LIN {X 0,Y 143.393,Z 441.137,A -85,B 0,C 180,E1 -24501.373,E2 -24501.373} C_VEL
LIN {X 0,Y 143.569,Z 442.834,A -85,B 0,C 180,E1 -24508.221,E2 -24508.221} C_VEL
LIN {X 0,Y 143.67,Z 443.783,A -85,B 0,C 180,E1 -24510.704,E2 -24510.704} C_VEL
LIN {X 0,Y 144.829,Z 446.872,A -85,B 0,C 180,E1 -24511.853,E2 -24511.853} C_VEL
LIN {X 0,Y 147.407,Z 450.098,A -85,B 0,C 180,E1 -24513.922,E2 -24513.922} C_VEL
LIN {X 0,Y 149.008,Z 453.626,A -85,B 0,C 180,E1 -24515.399,E2 -24515.399} C_VEL
LIN {X 0,Y 150.515,Z 455.827,A -85,B 0,C 180,E1 -24516.538,E2 -24516.538} C_VEL
LIN {X 0,Y 154.839,Z 465.074,A -85,B 0,C 180,E1 -24520.302,E2 -24520.302} C_VEL
LIN {X 0,Y 156.776,Z 470.615,A -85,B 0,C 180,E1 -24522.256,E2 -24522.256} C_VEL
LIN {X 0,Y 158.409,Z 477.402,A -85,B 0,C 180,E1 -24524.42,E2 -24524.42} C_VEL
LIN {X 0,Y 159.626,Z 487.108,A -85,B 0,C 180,E1 -24527.387,E2 -24527.387} C_VEL
LIN {X 0,Y 159.828,Z 498.246,A -85,B 0,C 180,E1 -24530.923,E2 -24530.923} C_VEL
LIN {X 0,Y 159.156,Z 506.693,A -85,B 0,C 180,E1 -24533.798,E2 -24533.798} C_VEL
LIN {X 0,Y 158.051,Z 513.314,A -85,B 0,C 180,E1 -24536.232,E2 -24536.232} C_VEL
LIN {X 0,Y 154.438,Z 521.15,A -85,B 0,C 180,E1 -24539.206,E2 -24539.206} C_VEL
LIN {X 0,Y 151.218,Z 527.693,A -85,B 0,C 180,E1 -24542.305,E2 -24542.305} C_VEL
LIN {X 0,Y 148.827,Z 532.196,A -85,B 0,C 180,E1 -24544.849,E2 -24544.849} C_VEL
LIN {X 0,Y 145.787,Z 537.691,A -85,B 0,C 180,E1 -24548.804,E2 -24548.804} C_VEL
LIN {X 0,Y 143.393,Z 542.02,A -85,B 0,C 180,E1 -24552.898,E2 -24552.898} C_VEL
LIN {X 0,Y 142.296,Z 544.395,A -85,B 0,C 180,E1 -24555.703,E2 -24555.703} C_VEL
LIN {X 0,Y 141.449,Z 546.201,A -85,B 0,C 180,E1 -24558.536,E2 -24558.536} C_VEL
LIN {X 0,Y 140.624,Z 548.663,A -85,B 0,C 180,E1 -24564.263,E2 -24564.263} C_VEL
LIN {X 0,Y 140.572,Z 549.418,A -85,B 0,C 180,E1 -24569.355,E2 -24569.355} C_VEL
LIN {X 0,Y 140.512,Z 549.259,A -85,B 0,C 180,E1 -24572.866,E2 -24572.866} C_VEL
LIN {X 0,Y 140.623,Z 548.664,A -85,B 0,C 180,E1 -24575.736,E2 -24575.736} C_VEL
LIN {X 0,Y 141.449,Z 546.201,A -85,B 0,C 180,E1 -24581.463,E2 -24581.463} C_VEL
LIN {X 0,Y 142.829,Z 543.242,A -85,B 0,C 180,E1 -24585.701,E2 -24585.701} C_VEL
LIN {X 0,Y 144.915,Z 539.247,A -85,B 0,C 180,E1 -24589.844,E2 -24589.844} C_VEL
LIN {X 0,Y 147.71,Z 534.114,A -85,B 0,C 180,E1 -24593.854,E2 -24593.854} C_VEL
LIN {X 0,Y 150.632,Z 528.852,A -85,B 0,C 180,E1 -24597.058,E2 -24597.058} C_VEL
LIN {X 0,Y 153.161,Z 523.745,A -85,B 0,C 180,E1 -24599.644,E2 -24599.644} C_VEL
LIN {X 0,Y 156.671,Z 516.577,A -85,B 0,C 180,E1 -24602.567,E2 -24602.567} C_VEL
LIN {X 0,Y 158.059,Z 513.317,A -85,B 0,C 180,E1 -24603.765,E2 -24603.765} C_VEL
LIN {X 0,Y 159.429,Z 504.825,A -85,B 0,C 180,E1 -24606.879,E2 -24606.879} C_VEL
LIN {X 0,Y 159.896,Z 494.943,A -85,B 0,C 180,E1 -24610.153,E2 -24610.153} C_VEL
LIN {X 0,Y 159.424,Z 485.143,A -85,B 0,C 180,E1 -24613.195,E2 -24613.195} C_VEL
LIN {X 0,Y 158.141,Z 476.083,A -85,B 0,C 180,E1 -24615.973,E2 -24615.973} C_VEL
LIN {X 0,Y 156.287,Z 468.906,A -85,B 0,C 180,E1 -24618.338,E2 -24618.338} C_VEL
LIN {X 0,Y 154.102,Z 463.522,A -85,B 0,C 180,E1 -24620.319,E2 -24620.319} C_VEL
LIN {X 0,Y 149.931,Z 454.821,A -85,B 0,C 180,E1 -24623.922,E2 -24623.922} C_VEL
LIN {X 0,Y 147.879,Z 451.476,A -85,B 0,C 180,E1 -24625.576,E2 -24625.576} C_VEL
LIN {X 0,Y 147.011,Z 449.414,A -85,B 0,C 180,E1 -24626.424,E2 -24626.424} C_VEL
LIN {X 0,Y 144.642,Z 446.551,A -85,B 0,C 180,E1 -24628.305,E2 -24628.305} C_VEL
LIN {X 0,Y 143.604,Z 443.405,A -85,B 0,C 180,E1 -24629.484,E2 -24629.484} C_VEL
LIN {X 0,Y 143.603,Z 443.398,A -85,B 0,C 180,E1 -24629.509,E2 -24629.509} C_VEL
LIN {X 0,Y 143.264,Z 443.023,A -85,B 0,C 180,E1 -24631.065,E2 -24631.065} C_VEL
LIN {X 0,Y 141.909,Z 442.618,A -85,B 0,C 180,E1 -24633.375,E2 -24633.375} C_VEL
LIN {X 0,Y 136.677,Z 441.804,A -85,B 0,C 180,E1 -24640.485,E2 -24640.485} C_VEL
LIN {X 0,Y 136.28,Z 441.543,A -85,B 0,C 180,E1 -24642.161,E2 -24642.161} C_VEL
LIN {X 0,Y 136.272,Z 441.029,A -85,B 0,C 180,E1 -24645.055,E2 -24645.055} C_VEL
LIN {X 0,Y 136.495,Z 440.983,A -85,B 0,C 180,E1 -24648.113,E2 -24648.113} C_VEL
LIN {X 0,Y 136.597,Z 440.97,A -85,B 0,C 180,E1 -24651.119,E2 -24651.119} C_VEL
LIN {X 0,Y 137.131,Z 440.87,A -85,B 0,C 180,E1 -24659.998,E2 -24659.998} C_VEL
LIN {X 0,Y 136.588,Z 440.963,A -85,B 0,C 180,E1 -24668.878,E2 -24668.878} C_VEL
LIN {X 0,Y 136.488,Z 440.983,A -85,B 0,C 180,E1 -24671.953,E2 -24671.953} C_VEL
LIN {X 0,Y 136.24,Z 441.013,A -85,B 0,C 180,E1 -24678.028,E2 -24678.028} C_VEL
LIN {X 0,Y 136.193,Z 441.017,A -85,B 0,C 180,E1 -24681.747,E2 -24681.747} C_VEL
LIN {X 0,Y 136.082,Z 441.071,A -85,B 0,C 180,E1 -24685.013,E2 -24685.013} C_VEL
LIN {X 0,Y 136.847,Z 443.396,A -85,B 0,C 180,E1 -24686.085,E2 -24686.085} C_VEL
LIN {X 0,Y 138.886,Z 445.821,A -85,B 0,C 180,E1 -24688.301,E2 -24688.301} C_VEL
LIN {X 0,Y 140.192,Z 446.89,A -85,B 0,C 180,E1 -24689.52,E2 -24689.52} C_VEL
LIN {X 0,Y 141.597,Z 449.723,A -85,B 0,C 180,E1 -24691.096,E2 -24691.096} C_VEL
LIN {X 0,Y 143.682,Z 451.967,A -85,B 0,C 180,E1 -24692.892,E2 -24692.892} C_VEL
LIN {X 0,Y 145.815,Z 455.547,A -85,B 0,C 180,E1 -24694.981,E2 -24694.981} C_VEL
LIN {X 0,Y 149.78,Z 462.277,A -85,B 0,C 180,E1 -24698.598,E2 -24698.598} C_VEL
LIN {X 0,Y 153.726,Z 470.155,A -85,B 0,C 180,E1 -24702.4,E2 -24702.4} C_VEL
LIN {X 0,Y 156.806,Z 478.027,A -85,B 0,C 180,E1 -24705.815,E2 -24705.815} C_VEL
LIN {X 0,Y 158.958,Z 485.07,A -85,B 0,C 180,E1 -24708.729,E2 -24708.729} C_VEL
LIN {X 0,Y 160.498,Z 491.796,A -85,B 0,C 180,E1 -24711.465,E2 -24711.465} C_VEL
LIN {X 0,Y 161.573,Z 498.214,A -85,B 0,C 180,E1 -24714.117,E2 -24714.117} C_VEL
LIN {X 0,Y 162.598,Z 505.476,A -85,B 0,C 180,E1 -24717.364,E2 -24717.364} C_VEL
LIN {X 0,Y 164.659,Z 513.088,A -85,B 0,C 180,E1 -24721.399,E2 -24721.399} C_VEL
LIN {X 0,Y 167.754,Z 519.177,A -85,B 0,C 180,E1 -24725.233,E2 -24725.233} C_VEL
LIN {X 0,Y 172.51,Z 524.998,A -85,B 0,C 180,E1 -24729.552,E2 -24729.552} C_VEL
LIN {X 0,Y 176.829,Z 528.462,A -85,B 0,C 180,E1 -24732.525,E2 -24732.525} C_VEL
LIN {X 0,Y 184.325,Z 532.617,A -85,B 0,C 180,E1 -24736.776,E2 -24736.776} C_VEL
LIN {X 0,Y 192.376,Z 535.547,A -85,B 0,C 180,E1 -24740.526,E2 -24740.526} C_VEL
LIN {X 0,Y 201.039,Z 537.521,A -85,B 0,C 180,E1 -24743.981,E2 -24743.981} C_VEL
LIN {X 0,Y 206.856,Z 538.379,A -85,B 0,C 180,E1 -24746.104,E2 -24746.104} C_VEL
LIN {X 0,Y 212.283,Z 538.785,A -85,B 0,C 180,E1 -24748.103,E2 -24748.103} C_VEL
LIN {X 0,Y 216.488,Z 538.826,A -85,B 0,C 180,E1 -24750,E2 -24750} C_VEL
LIN {X 0,Y 212.31,Z 538.784,A -85,B 0,C 180,E1 -24751.897,E2 -24751.897} C_VEL
LIN {X 0,Y 204.513,Z 538.092,A -85,B 0,C 180,E1 -24754.759,E2 -24754.759} C_VEL
LIN {X 0,Y 195.316,Z 536.345,A -85,B 0,C 180,E1 -24758.276,E2 -24758.276} C_VEL
LIN {X 0,Y 186.807,Z 533.661,A -85,B 0,C 180,E1 -24762.003,E2 -24762.003} C_VEL
LIN {X 0,Y 179.372,Z 530.065,A -85,B 0,C 180,E1 -24765.919,E2 -24765.919} C_VEL
LIN {X 0,Y 173.655,Z 526.039,A -85,B 0,C 180,E1 -24769.596,E2 -24769.596} C_VEL
LIN {X 0,Y 168.811,Z 520.752,A -85,B 0,C 180,E1 -24773.668,E2 -24773.668} C_VEL
LIN {X 0,Y 165.747,Z 515.636,A -85,B 0,C 180,E1 -24777.075,E2 -24777.075} C_VEL
LIN {X 0,Y 163.456,Z 509.289,A -85,B 0,C 180,E1 -24780.695,E2 -24780.695} C_VEL
LIN {X 0,Y 162.22,Z 503.336,A -85,B 0,C 180,E1 -24783.649,E2 -24783.649} C_VEL
LIN {X 0,Y 161.234,Z 495.681,A -85,B 0,C 180,E1 -24786.939,E2 -24786.939} C_VEL
LIN {X 0,Y 159.656,Z 487.905,A -85,B 0,C 180,E1 -24790.155,E2 -24790.155} C_VEL
LIN {X 0,Y 157.146,Z 479.075,A -85,B 0,C 180,E1 -24793.77,E2 -24793.77} C_VEL
LIN {X 0,Y 153.7,Z 470.237,A -85,B 0,C 180,E1 -24797.591,E2 -24797.591} C_VEL
LIN {X 0,Y 148.933,Z 460.739,A -85,B 0,C 180,E1 -24802.162,E2 -24802.162} C_VEL
LIN {X 0,Y 145.766,Z 455.541,A -85,B 0,C 180,E1 -24805.049,E2 -24805.049} C_VEL
LIN {X 0,Y 143.589,Z 451.797,A -85,B 0,C 180,E1 -24807.198,E2 -24807.198} C_VEL
LIN {X 0,Y 140.934,Z 448.683,A -85,B 0,C 180,E1 -24809.573,E2 -24809.573} C_VEL
LIN {X 0,Y 140.071,Z 446.555,A -85,B 0,C 180,E1 -24810.64,E2 -24810.64} C_VEL
LIN {X 0,Y 137.435,Z 444.32,A -85,B 0,C 180,E1 -24813.217,E2 -24813.217} C_VEL
LIN {X 0,Y 136.247,Z 441.933,A -85,B 0,C 180,E1 -24814.714,E2 -24814.714} C_VEL
LIN {X 0,Y 136.085,Z 441.023,A -85,B 0,C 180,E1 -24815.09,E2 -24815.09} C_VEL
LIN {X 0,Y 136.242,Z 441.007,A -85,B 0,C 180,E1 -24818.835,E2 -24818.835} C_VEL
LIN {X 0,Y 136.275,Z 440.999,A -85,B 0,C 180,E1 -24825.059,E2 -24825.059} C_VEL
LIN {X 0,Y 136.497,Z 440.982,A -85,B 0,C 180,E1 -24828.116,E2 -24828.116} C_VEL
LIN {X 0,Y 136.591,Z 440.963,A -85,B 0,C 180,E1 -24831.122,E2 -24831.122} C_VEL
LIN {X 0,Y 137.134,Z 440.87,A -85,B 0,C 180,E1 -24840.002,E2 -24840.002} C_VEL
LIN {X 0,Y 136.6,Z 440.97,A -85,B 0,C 180,E1 -24848.881,E2 -24848.881} C_VEL
LIN {X 0,Y 136.492,Z 440.986,A -85,B 0,C 180,E1 -24851.956,E2 -24851.956} C_VEL
LIN {X 0,Y 136.275,Z 441.029,A -85,B 0,C 180,E1 -24854.945,E2 -24854.945} C_VEL
LIN {X 0,Y 136.389,Z 442.204,A -85,B 0,C 180,E1 -24861.145,E2 -24861.145} C_VEL
LIN {X 0,Y 136.395,Z 443.172,A -85,B 0,C 180,E1 -24865.057,E2 -24865.057} C_VEL
LIN {X 0,Y 137.556,Z 446.287,A -85,B 0,C 180,E1 -24866.557,E2 -24866.557} C_VEL
LIN {X 0,Y 140.112,Z 449.358,A -85,B 0,C 180,E1 -24869.122,E2 -24869.122} C_VEL
LIN {X 0,Y 140.609,Z 450.141,A -85,B 0,C 180,E1 -24869.639,E2 -24869.639} C_VEL
LIN {X 0,Y 142.08,Z 453.455,A -85,B 0,C 180,E1 -24871.293,E2 -24871.293} C_VEL
LIN {X 0,Y 143.832,Z 455.753,A -85,B 0,C 180,E1 -24872.826,E2 -24872.826} C_VEL
LIN {X 0,Y 145.538,Z 459.421,A -85,B 0,C 180,E1 -24874.571,E2 -24874.571} C_VEL
LIN {X 0,Y 146.291,Z 460.539,A -85,B 0,C 180,E1 -24875.244,E2 -24875.244} C_VEL
LIN {X 0,Y 150.353,Z 470.127,A -85,B 0,C 180,E1 -24879.437,E2 -24879.437} C_VEL
LIN {X 0,Y 152.33,Z 476.964,A -85,B 0,C 180,E1 -24881.992,E2 -24881.992} C_VEL
LIN {X 0,Y 153.471,Z 485.376,A -85,B 0,C 180,E1 -24884.816,E2 -24884.816} C_VEL
LIN {X 0,Y 153.84,Z 493.755,A -85,B 0,C 180,E1 -24887.61,E2 -24887.61} C_VEL
LIN {X 0,Y 153.408,Z 503.934,A -85,B 0,C 180,E1 -24891.154,E2 -24891.154} C_VEL
LIN {X 0,Y 151.957,Z 513.094,A -85,B 0,C 180,E1 -24894.681,E2 -24894.681} C_VEL
LIN {X 0,Y 150.705,Z 516.362,A -85,B 0,C 180,E1 -24895.971,E2 -24895.971} C_VEL
LIN {X 0,Y 147.619,Z 522.314,A -85,B 0,C 180,E1 -24898.419,E2 -24898.419} C_VEL
LIN {X 0,Y 144.306,Z 528.638,A -85,B 0,C 180,E1 -24901.651,E2 -24901.651} C_VEL
LIN {X 0,Y 141.222,Z 533.9,A -85,B 0,C 180,E1 -24904.975,E2 -24904.975} C_VEL
LIN {X 0,Y 138.221,Z 539.034,A -85,B 0,C 180,E1 -24909.15,E2 -24909.15} C_VEL
LIN {X 0,Y 135.961,Z 543.029,A -85,B 0,C 180,E1 -24913.482,E2 -24913.482} C_VEL
LIN {X 0,Y 134.481,Z 545.989,A -85,B 0,C 180,E1 -24917.933,E2 -24917.933} C_VEL
LIN {X 0,Y 133.55,Z 548.452,A -85,B 0,C 180,E1 -24923.958,E2 -24923.958} C_VEL
LIN {X 0,Y 133.414,Z 549.047,A -85,B 0,C 180,E1 -24926.98,E2 -24926.98} C_VEL
LIN {X 0,Y 133.505,Z 549.208,A -85,B 0,C 180,E1 -24929.999,E2 -24929.999} C_VEL
LIN {X 0,Y 133.415,Z 549.048,A -85,B 0,C 180,E1 -24933.019,E2 -24933.019} C_VEL
LIN {X 0,Y 133.55,Z 548.452,A -85,B 0,C 180,E1 -24936.041,E2 -24936.041} C_VEL
LIN {X 0,Y 134.481,Z 545.989,A -85,B 0,C 180,E1 -24942.065,E2 -24942.065} C_VEL
LIN {X 0,Y 135.96,Z 543.03,A -85,B 0,C 180,E1 -24946.516,E2 -24946.516} C_VEL
LIN {X 0,Y 138.219,Z 539.035,A -85,B 0,C 180,E1 -24950.849,E2 -24950.849} C_VEL
LIN {X 0,Y 141.216,Z 533.901,A -85,B 0,C 180,E1 -24955.025,E2 -24955.025} C_VEL
LIN {X 0,Y 144.308,Z 528.64,A -85,B 0,C 180,E1 -24958.348,E2 -24958.348} C_VEL
LIN {X 0,Y 147.617,Z 522.316,A -85,B 0,C 180,E1 -24961.58,E2 -24961.58} C_VEL
LIN {X 0,Y 150.703,Z 516.365,A -85,B 0,C 180,E1 -24964.028,E2 -24964.028} C_VEL
LIN {X 0,Y 151.961,Z 513.096,A -85,B 0,C 180,E1 -24965.316,E2 -24965.316} C_VEL
LIN {X 0,Y 153.432,Z 503.887,A -85,B 0,C 180,E1 -24968.857,E2 -24968.857} C_VEL
LIN {X 0,Y 153.833,Z 493.811,A -85,B 0,C 180,E1 -24972.374,E2 -24972.374} C_VEL
LIN {X 0,Y 153.466,Z 485.366,A -85,B 0,C 180,E1 -24975.188,E2 -24975.188} C_VEL
LIN {X 0,Y 152.317,Z 477.003,A -85,B 0,C 180,E1 -24978.004,E2 -24978.004} C_VEL
LIN {X 0,Y 150.358,Z 470.111,A -85,B 0,C 180,E1 -24980.565,E2 -24980.565} C_VEL
LIN {X 0,Y 146.266,Z 460.462,A -85,B 0,C 180,E1 -24984.787,E2 -24984.787} C_VEL
LIN {X 0,Y 144.146,Z 456.557,A -85,B 0,C 180,E1 -24986.838,E2 -24986.838} C_VEL
LIN {X 0,Y 143.387,Z 455.024,A -85,B 0,C 180,E1 -24987.58,E2 -24987.58} C_VEL
LIN {X 0,Y 141.186,Z 451.788,A -85,B 0,C 180,E1 -24989.63,E2 -24989.63} C_VEL
LIN {X 0,Y 140.254,Z 449.367,A -85,B 0,C 180,E1 -24990.773,E2 -24990.773} C_VEL
LIN {X 0,Y 137.632,Z 446.44,A -85,B 0,C 180,E1 -24993.357,E2 -24993.357} C_VEL
LIN {X 0,Y 136.433,Z 443.429,A -85,B 0,C 180,E1 -24994.849,E2 -24994.849} C_VEL
LIN {X 0,Y 136.355,Z 442.979,A -85,B 0,C 180,E1 -24995.241,E2 -24995.241} C_VEL
LIN {X 0,Y 136.368,Z 442.185,A -85,B 0,C 180,E1 -24998.851,E2 -24998.851} C_VEL
LIN {X 0,Y 136.28,Z 441.543,A -85,B 0,C 180,E1 -25002.161,E2 -25002.161} C_VEL
LIN {X 0,Y 135.521,Z 441.297,A -85,B 0,C 180,E1 -25004.629,E2 -25004.629} C_VEL
LIN {X 0,Y 133.951,Z 441.34,A -85,B 0,C 180,E1 -25007.072,E2 -25007.072} C_VEL
LIN {X 0,Y 129.756,Z 441.823,A -85,B 0,C 180,E1 -25013.816,E2 -25013.816} C_VEL
LIN {X 0,Y 129.561,Z 441.841,A -85,B 0,C 180,E1 -25015.588,E2 -25015.588} C_VEL
LIN {X 0,Y 130.086,Z 441.745,A -85,B 0,C 180,E1 -25019.998,E2 -25019.998} C_VEL
LIN {X 0,Y 129.514,Z 441.842,A -85,B 0,C 180,E1 -25029.367,E2 -25029.367} C_VEL
LIN {X 0,Y 129.39,Z 441.868,A -85,B 0,C 180,E1 -25032.547,E2 -25032.547} C_VEL
LIN {X 0,Y 129.227,Z 442.093,A -85,B 0,C 180,E1 -25037.505,E2 -25037.505} C_VEL
LIN {X 0,Y 129.982,Z 444.418,A -85,B 0,C 180,E1 -25039.133,E2 -25039.133} C_VEL
LIN {X 0,Y 132.518,Z 447.116,A -85,B 0,C 180,E1 -25042.908,E2 -25042.908} C_VEL
LIN {X 0,Y 133.418,Z 447.725,A -85,B 0,C 180,E1 -25043.989,E2 -25043.989} C_VEL
LIN {X 0,Y 134.689,Z 450.544,A -85,B 0,C 180,E1 -25045.911,E2 -25045.911} C_VEL
LIN {X 0,Y 136.266,Z 452.208,A -85,B 0,C 180,E1 -25047.655,E2 -25047.655} C_VEL
LIN {X 0,Y 138.6,Z 455.974,A -85,B 0,C 180,E1 -25050.467,E2 -25050.467} C_VEL
LIN {X 0,Y 139.949,Z 457.473,A -85,B 0,C 180,E1 -25051.821,E2 -25051.821} C_VEL
LIN {X 0,Y 144.358,Z 465.277,A -85,B 0,C 180,E1 -25056.609,E2 -25056.609} C_VEL
LIN {X 0,Y 147.935,Z 472.663,A -85,B 0,C 180,E1 -25060.528,E2 -25060.528} C_VEL
LIN {X 0,Y 150.939,Z 480.552,A -85,B 0,C 180,E1 -25064.299,E2 -25064.299} C_VEL
LIN {X 0,Y 153.326,Z 489.067,A -85,B 0,C 180,E1 -25068.131,E2 -25068.131} C_VEL
LIN {X 0,Y 154.949,Z 497.906,A -85,B 0,C 180,E1 -25072.082,E2 -25072.082} C_VEL
LIN {X 0,Y 155.807,Z 506.276,A -85,B 0,C 180,E1 -25076.024,E2 -25076.024} C_VEL
LIN {X 0,Y 157.299,Z 513.318,A -85,B 0,C 180,E1 -25079.915,E2 -25079.915} C_VEL
LIN {X 0,Y 159.806,Z 519.439,A -85,B 0,C 180,E1 -25083.911,E2 -25083.911} C_VEL
LIN {X 0,Y 164.077,Z 525.325,A -85,B 0,C 180,E1 -25088.494,E2 -25088.494} C_VEL
LIN {X 0,Y 167.934,Z 528.774,A -85,B 0,C 180,E1 -25091.599,E2 -25091.599} C_VEL
LIN {X 0,Y 174.984,Z 532.897,A -85,B 0,C 180,E1 -25096.056,E2 -25096.056} C_VEL
LIN {X 0,Y 180.186,Z 535.032,A -85,B 0,C 180,E1 -25098.755,E2 -25098.755} C_VEL
LIN {X 0,Y 190.977,Z 537.733,A -85,B 0,C 180,E1 -25103.506,E2 -25103.506} C_VEL
LIN {X 0,Y 197.369,Z 538.659,A -85,B 0,C 180,E1 -25105.917,E2 -25105.917} C_VEL
LIN {X 0,Y 203.898,Z 539.101,A -85,B 0,C 180,E1 -25108.29,E2 -25108.29} C_VEL
LIN {X 0,Y 208.174,Z 539.069,A -85,B 0,C 180,E1 -25110,E2 -25110} C_VEL
LIN {X 0,Y 203.184,Z 539.054,A -85,B 0,C 180,E1 -25111.983,E2 -25111.983} C_VEL
LIN {X 0,Y 197.29,Z 538.649,A -85,B 0,C 180,E1 -25114.123,E2 -25114.123} C_VEL
LIN {X 0,Y 185.008,Z 536.433,A -85,B 0,C 180,E1 -25119.012,E2 -25119.012} C_VEL
LIN {X 0,Y 179.381,Z 534.763,A -85,B 0,C 180,E1 -25121.635,E2 -25121.635} C_VEL
LIN {X 0,Y 172.472,Z 531.671,A -85,B 0,C 180,E1 -25125.439,E2 -25125.439} C_VEL
LIN {X 0,Y 165.148,Z 526.409,A -85,B 0,C 180,E1 -25130.577,E2 -25130.577} C_VEL
LIN {X 0,Y 160.856,Z 521.236,A -85,B 0,C 180,E1 -25134.778,E2 -25134.778} C_VEL
LIN {X 0,Y 158.352,Z 516.365,A -85,B 0,C 180,E1 -25138.192,E2 -25138.192} C_VEL
LIN {X 0,Y 156.393,Z 509.827,A -85,B 0,C 180,E1 -25142.104,E2 -25142.104} C_VEL
LIN {X 0,Y 155.368,Z 502.005,A -85,B 0,C 180,E1 -25146.019,E2 -25146.019} C_VEL
LIN {X 0,Y 154.77,Z 496.619,A -85,B 0,C 180,E1 -25148.5,E2 -25148.5} C_VEL
LIN {X 0,Y 152.849,Z 487.303,A -85,B 0,C 180,E1 -25152.638,E2 -25152.638} C_VEL
LIN {X 0,Y 150.411,Z 479.196,A -85,B 0,C 180,E1 -25156.331,E2 -25156.331} C_VEL
LIN {X 0,Y 147.044,Z 470.89,A -85,B 0,C 180,E1 -25160.417,E2 -25160.417} C_VEL
LIN {X 0,Y 142.649,Z 462.223,A -85,B 0,C 180,E1 -25165.254,E2 -25165.254} C_VEL
LIN {X 0,Y 139.958,Z 457.442,A -85,B 0,C 180,E1 -25168.182,E2 -25168.182} C_VEL
LIN {X 0,Y 138.562,Z 455.937,A -85,B 0,C 180,E1 -25169.571,E2 -25169.571} C_VEL
LIN {X 0,Y 136.097,Z 452.067,A -85,B 0,C 180,E1 -25172.516,E2 -25172.516} C_VEL
LIN {X 0,Y 134.091,Z 449.489,A -85,B 0,C 180,E1 -25174.901,E2 -25174.901} C_VEL
LIN {X 0,Y 133.205,Z 447.512,A -85,B 0,C 180,E1 -25176.28,E2 -25176.28} C_VEL
LIN {X 0,Y 130.402,Z 445.11,A -85,B 0,C 180,E1 -25180.112,E2 -25180.112} C_VEL
LIN {X 0,Y 129.475,Z 443.087,A -85,B 0,C 180,E1 -25181.917,E2 -25181.917} C_VEL
LIN {X 0,Y 129.183,Z 441.894,A -85,B 0,C 180,E1 -25182.795,E2 -25182.795} C_VEL
LIN {X 0,Y 129.416,Z 441.865,A -85,B 0,C 180,E1 -25187.822,E2 -25187.822} C_VEL
LIN {X 0,Y 129.517,Z 441.842,A -85,B 0,C 180,E1 -25190.633,E2 -25190.633} C_VEL
LIN {X 0,Y 130.089,Z 441.745,A -85,B 0,C 180,E1 -25200.002,E2 -25200.002} C_VEL
LIN {X 0,Y 129.524,Z 441.852,A -85,B 0,C 180,E1 -25209.37,E2 -25209.37} C_VEL
LIN {X 0,Y 129.394,Z 441.868,A -85,B 0,C 180,E1 -25212.55,E2 -25212.55} C_VEL
LIN {X 0,Y 129.304,Z 442.792,A -85,B 0,C 180,E1 -25217.192,E2 -25217.192} C_VEL
LIN {X 0,Y 130.413,Z 445.846,A -85,B 0,C 180,E1 -25219.378,E2 -25219.378} C_VEL
LIN {X 0,Y 133.368,Z 449.231,A -85,B 0,C 180,E1 -25223.487,E2 -25223.487} C_VEL
LIN {X 0,Y 133.838,Z 449.932,A -85,B 0,C 180,E1 -25224.119,E2 -25224.119} C_VEL
LIN {X 0,Y 135.258,Z 453.28,A -85,B 0,C 180,E1 -25226.212,E2 -25226.212} C_VEL
LIN {X 0,Y 137.402,Z 456.073,A -85,B 0,C 180,E1 -25228.552,E2 -25228.552} C_VEL
LIN {X 0,Y 138.83,Z 459.389,A -85,B 0,C 180,E1 -25230.415,E2 -25230.415} C_VEL
LIN {X 0,Y 140.009,Z 461.026,A -85,B 0,C 180,E1 -25231.64,E2 -25231.64} C_VEL
LIN {X 0,Y 141.231,Z 464.087,A -85,B 0,C 180,E1 -25233.19,E2 -25233.19} C_VEL
LIN {X 0,Y 142.564,Z 466.668,A -85,B 0,C 180,E1 -25234.602,E2 -25234.602} C_VEL
LIN {X 0,Y 145.848,Z 475.588,A -85,B 0,C 180,E1 -25238.789,E2 -25238.789} C_VEL
LIN {X 0,Y 147.264,Z 481.982,A -85,B 0,C 180,E1 -25241.364,E2 -25241.364} C_VEL
LIN {X 0,Y 147.897,Z 489.71,A -85,B 0,C 180,E1 -25244.137,E2 -25244.137} C_VEL
LIN {X 0,Y 147.828,Z 498.018,A -85,B 0,C 180,E1 -25247.135,E2 -25247.135} C_VEL
LIN {X 0,Y 147.28,Z 505.011,A -85,B 0,C 180,E1 -25249.776,E2 -25249.776} C_VEL
LIN {X 0,Y 145.909,Z 512.871,A -85,B 0,C 180,E1 -25252.98,E2 -25252.98} C_VEL
LIN {X 0,Y 144.824,Z 516.149,A -85,B 0,C 180,E1 -25254.385,E2 -25254.385} C_VEL
LIN {X 0,Y 141.592,Z 522.102,A -85,B 0,C 180,E1 -25256.907,E2 -25256.907} C_VEL
LIN {X 0,Y 138.345,Z 527.892,A -85,B 0,C 180,E1 -25259.924,E2 -25259.924} C_VEL
LIN {X 0,Y 136.103,Z 531.774,A -85,B 0,C 180,E1 -25262.307,E2 -25262.307} C_VEL
LIN {X 0,Y 132.597,Z 537.267,A -85,B 0,C 180,E1 -25266.576,E2 -25266.576} C_VEL
LIN {X 0,Y 129.821,Z 541.595,A -85,B 0,C 180,E1 -25271.045,E2 -25271.045} C_VEL
LIN {X 0,Y 128.538,Z 543.971,A -85,B 0,C 180,E1 -25274.134,E2 -25274.134} C_VEL
LIN {X 0,Y 127.51,Z 545.776,A -85,B 0,C 180,E1 -25277.263,E2 -25277.263} C_VEL
LIN {X 0,Y 126.472,Z 548.24,A -85,B 0,C 180,E1 -25283.618,E2 -25283.618} C_VEL
LIN {X 0,Y 126.317,Z 548.836,A -85,B 0,C 180,E1 -25286.81,E2 -25286.81} C_VEL
LIN {X 0,Y 126.424,Z 548.997,A -85,B 0,C 180,E1 -25289.999,E2 -25289.999} C_VEL
LIN {X 0,Y 126.318,Z 548.836,A -85,B 0,C 180,E1 -25293.189,E2 -25293.189} C_VEL
LIN {X 0,Y 126.471,Z 548.24,A -85,B 0,C 180,E1 -25296.38,E2 -25296.38} C_VEL
LIN {X 0,Y 127.509,Z 545.777,A -85,B 0,C 180,E1 -25302.736,E2 -25302.736} C_VEL
LIN {X 0,Y 129.133,Z 542.817,A -85,B 0,C 180,E1 -25307.417,E2 -25307.417} C_VEL
LIN {X 0,Y 131.579,Z 538.823,A -85,B 0,C 180,E1 -25311.955,E2 -25311.955} C_VEL
LIN {X 0,Y 134.796,Z 533.689,A -85,B 0,C 180,E1 -25316.305,E2 -25316.305} C_VEL
LIN {X 0,Y 137.385,Z 529.617,A -85,B 0,C 180,E1 -25319.051,E2 -25319.051} C_VEL
LIN {X 0,Y 140.772,Z 523.619,A -85,B 0,C 180,E1 -25322.373,E2 -25322.373} C_VEL
LIN {X 0,Y 144.023,Z 517.78,A -85,B 0,C 180,E1 -25324.985,E2 -25324.985} C_VEL
LIN {X 0,Y 145.464,Z 514.517,A -85,B 0,C 180,E1 -25326.287,E2 -25326.287} C_VEL
LIN {X 0,Y 147.02,Z 506.725,A -85,B 0,C 180,E1 -25329.524,E2 -25329.524} C_VEL
LIN {X 0,Y 147.639,Z 500.871,A -85,B 0,C 180,E1 -25331.791,E2 -25331.791} C_VEL
LIN {X 0,Y 147.941,Z 493.393,A -85,B 0,C 180,E1 -25334.553,E2 -25334.553} C_VEL
LIN {X 0,Y 147.564,Z 484.85,A -85,B 0,C 180,E1 -25337.625,E2 -25337.625} C_VEL
LIN {X 0,Y 146.59,Z 478.323,A -85,B 0,C 180,E1 -25340.091,E2 -25340.091} C_VEL
LIN {X 0,Y 144.213,Z 470.828,A -85,B 0,C 180,E1 -25343.344,E2 -25343.344} C_VEL
LIN {X 0,Y 142.17,Z 465.659,A -85,B 0,C 180,E1 -25345.867,E2 -25345.867} C_VEL
LIN {X 0,Y 140.573,Z 462.676,A -85,B 0,C 180,E1 -25347.573,E2 -25347.573} C_VEL
LIN {X 0,Y 140.021,Z 460.986,A -85,B 0,C 180,E1 -25348.363,E2 -25348.363} C_VEL
LIN {X 0,Y 138.262,Z 458.277,A -85,B 0,C 180,E1 -25350.289,E2 -25350.289} C_VEL
LIN {X 0,Y 137.042,Z 455.312,A -85,B 0,C 180,E1 -25351.888,E2 -25351.888} C_VEL
LIN {X 0,Y 134.638,Z 452.159,A -85,B 0,C 180,E1 -25354.593,E2 -25354.593} C_VEL
LIN {X 0,Y 133.536,Z 449.278,A -85,B 0,C 180,E1 -25356.339,E2 -25356.339} C_VEL
LIN {X 0,Y 130.586,Z 446.142,A -85,B 0,C 180,E1 -25360.342,E2 -25360.342} C_VEL
LIN {X 0,Y 129.409,Z 443.263,A -85,B 0,C 180,E1 -25362.517,E2 -25362.517} C_VEL
LIN {X 0,Y 129.257,Z 442.518,A -85,B 0,C 180,E1 -25363.005,E2 -25363.005} C_VEL
LIN {X 0,Y 129.415,Z 441.866,A -85,B 0,C 180,E1 -25367.818,E2 -25367.818} C_VEL
LIN {X 0,Y 129.521,Z 441.853,A -85,B 0,C 180,E1 -25370.63,E2 -25370.63} C_VEL
LIN {X 0,Y 129.561,Z 441.841,A -85,B 0,C 180,E1 -25375.588,E2 -25375.588} C_VEL
LIN {X 0,Y 129.354,Z 441.974,A -85,B 0,C 180,E1 -25377.321,E2 -25377.321} C_VEL
LIN {X 0,Y 128.656,Z 442.345,A -85,B 0,C 180,E1 -25379.034,E2 -25379.034} C_VEL
LIN {X 0,Y 126.526,Z 443.563,A -85,B 0,C 180,E1 -25382.434,E2 -25382.434} C_VEL
LIN {X 0,Y 124.538,Z 445.099,A -85,B 0,C 180,E1 -25385.944,E2 -25385.944} C_VEL
LIN {X 0,Y 124.03,Z 446.208,A -85,B 0,C 180,E1 -25388.663,E2 -25388.663} C_VEL
LIN {X 0,Y 124.174,Z 446.534,A -85,B 0,C 180,E1 -25389.574,E2 -25389.574} C_VEL
LIN {X 0,Y 127.019,Z 448.867,A -85,B 0,C 180,E1 -25396.575,E2 -25396.575} C_VEL
LIN {X 0,Y 128.029,Z 451.495,A -85,B 0,C 180,E1 -25399.02,E2 -25399.02} C_VEL
LIN {X 0,Y 130.089,Z 453.655,A -85,B 0,C 180,E1 -25402.219,E2 -25402.219} C_VEL
LIN {X 0,Y 134.078,Z 459.811,A -85,B 0,C 180,E1 -25408.146,E2 -25408.146} C_VEL
LIN {X 0,Y 136.408,Z 463.346,A -85,B 0,C 180,E1 -25411.01,E2 -25411.01} C_VEL
LIN {X 0,Y 140.865,Z 472.251,A -85,B 0,C 180,E1 -25416.775,E2 -25416.775} C_VEL
LIN {X 0,Y 143.775,Z 479.353,A -85,B 0,C 180,E1 -25420.778,E2 -25420.778} C_VEL
LIN {X 0,Y 145.93,Z 486.193,A -85,B 0,C 180,E1 -25424.288,E2 -25424.288} C_VEL
LIN {X 0,Y 147.472,Z 492.638,A -85,B 0,C 180,E1 -25427.449,E2 -25427.449} C_VEL
LIN {X 0,Y 148.627,Z 500.019,A -85,B 0,C 180,E1 -25431.034,E2 -25431.034} C_VEL
LIN {X 0,Y 149.123,Z 506.297,A -85,B 0,C 180,E1 -25434.159,E2 -25434.159} C_VEL
LIN {X 0,Y 150.119,Z 513.507,A -85,B 0,C 180,E1 -25438.279,E2 -25438.279} C_VEL
LIN {X 0,Y 152.08,Z 519.696,A -85,B 0,C 180,E1 -25442.477,E2 -25442.477} C_VEL
LIN {X 0,Y 154.528,Z 523.992,A -85,B 0,C 180,E1 -25445.839,E2 -25445.839} C_VEL
LIN {X 0,Y 159.451,Z 529.251,A -85,B 0,C 180,E1 -25450.771,E2 -25450.771} C_VEL
LIN {X 0,Y 165.816,Z 533.173,A -85,B 0,C 180,E1 -25455.268,E2 -25455.268} C_VEL
LIN {X 0,Y 171.957,Z 535.704,A -85,B 0,C 180,E1 -25458.775,E2 -25458.775} C_VEL
LIN {X 0,Y 177.639,Z 537.319,A -85,B 0,C 180,E1 -25461.516,E2 -25461.516} C_VEL
LIN {X 0,Y 187.713,Z 538.944,A -85,B 0,C 180,E1 -25465.706,E2 -25465.706} C_VEL
LIN {X 0,Y 196.81,Z 539.398,A -85,B 0,C 180,E1 -25468.999,E2 -25468.999} C_VEL
LIN {X 0,Y 199.44,Z 539.324,A -85,B 0,C 180,E1 -25470,E2 -25470} C_VEL
LIN {X 0,Y 193.787,Z 539.332,A -85,B 0,C 180,E1 -25472.079,E2 -25472.079} C_VEL
LIN {X 0,Y 183.692,Z 538.4,A -85,B 0,C 180,E1 -25475.887,E2 -25475.887} C_VEL
LIN {X 0,Y 176.118,Z 536.912,A -85,B 0,C 180,E1 -25479.185,E2 -25479.185} C_VEL
LIN {X 0,Y 170.709,Z 535.319,A -85,B 0,C 180,E1 -25481.879,E2 -25481.879} C_VEL
LIN {X 0,Y 161.947,Z 531.031,A -85,B 0,C 180,E1 -25487.311,E2 -25487.311} C_VEL
LIN {X 0,Y 157.603,Z 527.614,A -85,B 0,C 180,E1 -25490.901,E2 -25490.901} C_VEL
LIN {X 0,Y 153.2,Z 521.906,A -85,B 0,C 180,E1 -25495.836,E2 -25495.836} C_VEL
LIN {X 0,Y 150.703,Z 516.003,A -85,B 0,C 180,E1 -25500.121,E2 -25500.121} C_VEL
LIN {X 0,Y 149.454,Z 510.214,A -85,B 0,C 180,E1 -25503.717,E2 -25503.717} C_VEL
LIN {X 0,Y 148.828,Z 502.248,A -85,B 0,C 180,E1 -25507.871,E2 -25507.871} C_VEL
LIN {X 0,Y 147.903,Z 495.231,A -85,B 0,C 180,E1 -25511.321,E2 -25511.321} C_VEL
LIN {X 0,Y 146.373,Z 487.853,A -85,B 0,C 180,E1 -25514.914,E2 -25514.914} C_VEL
LIN {X 0,Y 144.379,Z 481.198,A -85,B 0,C 180,E1 -25518.307,E2 -25518.307} C_VEL
LIN {X 0,Y 141.788,Z 474.538,A -85,B 0,C 180,E1 -25521.897,E2 -25521.897} C_VEL
LIN {X 0,Y 138.532,Z 467.648,A -85,B 0,C 180,E1 -25526.081,E2 -25526.081} C_VEL
LIN {X 0,Y 136.414,Z 463.329,A -85,B 0,C 180,E1 -25528.991,E2 -25528.991} C_VEL
LIN {X 0,Y 132.977,Z 458.209,A -85,B 0,C 180,E1 -25533.307,E2 -25533.307} C_VEL
LIN {X 0,Y 129.821,Z 453.442,A -85,B 0,C 180,E1 -25538.151,E2 -25538.151} C_VEL
LIN {X 0,Y 127.553,Z 450.628,A -85,B 0,C 180,E1 -25541.947,E2 -25541.947} C_VEL
LIN {X 0,Y 126.998,Z 448.702,A -85,B 0,C 180,E1 -25543.526,E2 -25543.526} C_VEL
LIN {X 0,Y 123.207,Z 443.52,A -85,B 0,C 180,E1 -25560.002,E2 -25560.002} C_VEL
LIN {X 0,Y 124.236,Z 446.606,A -85,B 0,C 180,E1 -25568.951,E2 -25568.951} C_VEL
LIN {X 0,Y 127.16,Z 449.398,A -85,B 0,C 180,E1 -25576.147,E2 -25576.147} C_VEL
LIN {X 0,Y 128.333,Z 452.712,A -85,B 0,C 180,E1 -25578.977,E2 -25578.977} C_VEL
LIN {X 0,Y 130.997,Z 456.056,A -85,B 0,C 180,E1 -25582.996,E2 -25582.996} C_VEL
LIN {X 0,Y 132.203,Z 459.191,A -85,B 0,C 180,E1 -25585.171,E2 -25585.171} C_VEL
LIN {X 0,Y 133.847,Z 461.592,A -85,B 0,C 180,E1 -25587.352,E2 -25587.352} C_VEL
LIN {X 0,Y 135.325,Z 465.194,A -85,B 0,C 180,E1 -25589.564,E2 -25589.564} C_VEL
LIN {X 0,Y 136.242,Z 466.568,A -85,B 0,C 180,E1 -25590.606,E2 -25590.606} C_VEL
LIN {X 0,Y 139.04,Z 473.933,A -85,B 0,C 180,E1 -25594.746,E2 -25594.746} C_VEL
LIN {X 0,Y 140.883,Z 479.813,A -85,B 0,C 180,E1 -25597.671,E2 -25597.671} C_VEL
LIN {X 0,Y 141.926,Z 485.365,A -85,B 0,C 180,E1 -25600.074,E2 -25600.074} C_VEL
LIN {X 0,Y 142.247,Z 494.818,A -85,B 0,C 180,E1 -25603.767,E2 -25603.767} C_VEL
LIN {X 0,Y 141.451,Z 504.459,A -85,B 0,C 180,E1 -25607.592,E2 -25607.592} C_VEL
LIN {X 0,Y 139.95,Z 512.646,A -85,B 0,C 180,E1 -25611.117,E2 -25611.117} C_VEL
LIN {X 0,Y 138.985,Z 515.933,A -85,B 0,C 180,E1 -25612.642,E2 -25612.642} C_VEL
LIN {X 0,Y 135.676,Z 521.889,A -85,B 0,C 180,E1 -25615.264,E2 -25615.264} C_VEL
LIN {X 0,Y 131.829,Z 528.286,A -85,B 0,C 180,E1 -25618.74,E2 -25618.74} C_VEL
LIN {X 0,Y 128.463,Z 533.476,A -85,B 0,C 180,E1 -25622.288,E2 -25622.288} C_VEL
LIN {X 0,Y 125,Z 538.609,A -85,B 0,C 180,E1 -25626.823,E2 -25626.823} C_VEL
LIN {X 0,Y 122.328,Z 542.603,A -85,B 0,C 180,E1 -25631.579,E2 -25631.579} C_VEL
LIN {X 0,Y 120.57,Z 545.564,A -85,B 0,C 180,E1 -25636.516,E2 -25636.516} C_VEL
LIN {X 0,Y 119.418,Z 548.029,A -85,B 0,C 180,E1 -25643.24,E2 -25643.24} C_VEL
LIN {X 0,Y 119.232,Z 548.625,A -85,B 0,C 180,E1 -25646.62,E2 -25646.62} C_VEL
LIN {X 0,Y 119.334,Z 548.786,A -85,B 0,C 180,E1 -25649.999,E2 -25649.999} C_VEL
LIN {X 0,Y 119.232,Z 548.625,A -85,B 0,C 180,E1 -25653.378,E2 -25653.378} C_VEL
LIN {X 0,Y 119.417,Z 548.029,A -85,B 0,C 180,E1 -25656.759,E2 -25656.759} C_VEL
LIN {X 0,Y 120.569,Z 545.565,A -85,B 0,C 180,E1 -25663.482,E2 -25663.482} C_VEL
LIN {X 0,Y 122.327,Z 542.604,A -85,B 0,C 180,E1 -25668.419,E2 -25668.419} C_VEL
LIN {X 0,Y 124.998,Z 538.611,A -85,B 0,C 180,E1 -25673.176,E2 -25673.176} C_VEL
LIN {X 0,Y 128.457,Z 533.478,A -85,B 0,C 180,E1 -25677.712,E2 -25677.712} C_VEL
LIN {X 0,Y 131.828,Z 528.287,A -85,B 0,C 180,E1 -25681.26,E2 -25681.26} C_VEL
LIN {X 0,Y 135.674,Z 521.892,A -85,B 0,C 180,E1 -25684.735,E2 -25684.735} C_VEL
LIN {X 0,Y 138.981,Z 515.935,A -85,B 0,C 180,E1 -25687.358,E2 -25687.358} C_VEL
LIN {X 0,Y 140.342,Z 510.875,A -85,B 0,C 180,E1 -25689.678,E2 -25689.678} C_VEL
LIN {X 0,Y 141.461,Z 504.445,A -85,B 0,C 180,E1 -25692.412,E2 -25692.412} C_VEL
LIN {X 0,Y 142.222,Z 493.603,A -85,B 0,C 180,E1 -25696.697,E2 -25696.697} C_VEL
LIN {X 0,Y 141.924,Z 485.369,A -85,B 0,C 180,E1 -25699.926,E2 -25699.926} C_VEL
LIN {X 0,Y 140.892,Z 479.792,A -85,B 0,C 180,E1 -25702.332,E2 -25702.332} C_VEL
LIN {X 0,Y 139.04,Z 473.932,A -85,B 0,C 180,E1 -25705.254,E2 -25705.254} C_VEL
LIN {X 0,Y 137.456,Z 469.838,A -85,B 0,C 180,E1 -25707.528,E2 -25707.528} C_VEL
LIN {X 0,Y 135.943,Z 466.119,A -85,B 0,C 180,E1 -25709.73,E2 -25709.73} C_VEL
LIN {X 0,Y 134.286,Z 462.9,A -85,B 0,C 180,E1 -25711.897,E2 -25711.897} C_VEL
LIN {X 0,Y 133.852,Z 461.575,A -85,B 0,C 180,E1 -25712.649,E2 -25712.649} C_VEL
LIN {X 0,Y 131.743,Z 458.243,A -85,B 0,C 180,E1 -25715.578,E2 -25715.578} C_VEL
LIN {X 0,Y 130.696,Z 455.49,A -85,B 0,C 180,E1 -25717.47,E2 -25717.47} C_VEL
LIN {X 0,Y 127.941,Z 451.951,A -85,B 0,C 180,E1 -25721.793,E2 -25721.793} C_VEL
LIN {X 0,Y 127.141,Z 449.215,A -85,B 0,C 180,E1 -25723.954,E2 -25723.954} C_VEL
LIN {X 0,Y 123.292,Z 445.083,A -85,B 0,C 180,E1 -25735.912,E2 -25735.912} C_VEL
LIN {X 0,Y 123.193,Z 443.548,A -85,B 0,C 180,E1 -25739.998,E2 -25739.998} C_VEL
LIN {X 0,Y 124.174,Z 446.534,A -85,B 0,C 180,E1 -25749.574,E2 -25749.574} C_VEL
LIN {X 0,Y 124.82,Z 448.177,A -85,B 0,C 180,E1 -25752.165,E2 -25752.165} C_VEL
LIN {X 0,Y 125.361,Z 450.854,A -85,B 0,C 180,E1 -25754.584,E2 -25754.584} C_VEL
LIN {X 0,Y 126.862,Z 459.241,A -85,B 0,C 180,E1 -25760.782,E2 -25760.782} C_VEL
LIN {X 0,Y 127.65,Z 460.847,A -85,B 0,C 180,E1 -25762.401,E2 -25762.401} C_VEL
LIN {X 0,Y 130.551,Z 465.593,A -85,B 0,C 180,E1 -25767.229,E2 -25767.229} C_VEL
LIN {X 0,Y 132.531,Z 469.039,A -85,B 0,C 180,E1 -25770.248,E2 -25770.248} C_VEL
LIN {X 0,Y 135.465,Z 475.455,A -85,B 0,C 180,E1 -25774.796,E2 -25774.796} C_VEL
LIN {X 0,Y 137.736,Z 481.031,A -85,B 0,C 180,E1 -25778.297,E2 -25778.297} C_VEL
LIN {X 0,Y 140.046,Z 488.623,A -85,B 0,C 180,E1 -25782.644,E2 -25782.644} C_VEL
LIN {X 0,Y 141.668,Z 496.557,A -85,B 0,C 180,E1 -25786.897,E2 -25786.897} C_VEL
LIN {X 0,Y 142.61,Z 505.278,A -85,B 0,C 180,E1 -25791.54,E2 -25791.54} C_VEL
LIN {X 0,Y 143.153,Z 513.804,A -85,B 0,C 180,E1 -25796.571,E2 -25796.571} C_VEL
LIN {X 0,Y 144.593,Z 520.104,A -85,B 0,C 180,E1 -25801.03,E2 -25801.03} C_VEL
LIN {X 0,Y 147.083,Z 525.068,A -85,B 0,C 180,E1 -25805.209,E2 -25805.209} C_VEL
LIN {X 0,Y 150.434,Z 529.066,A -85,B 0,C 180,E1 -25809.121,E2 -25809.121} C_VEL
LIN {X 0,Y 154.509,Z 532.296,A -85,B 0,C 180,E1 -25812.781,E2 -25812.781} C_VEL
LIN {X 0,Y 161.421,Z 535.603,A -85,B 0,C 180,E1 -25817.427,E2 -25817.427} C_VEL
LIN {X 0,Y 170.288,Z 538.044,A -85,B 0,C 180,E1 -25822.09,E2 -25822.09} C_VEL
LIN {X 0,Y 178.053,Z 539.228,A -85,B 0,C 180,E1 -25825.473,E2 -25825.473} C_VEL
LIN {X 0,Y 184.194,Z 539.617,A -85,B 0,C 180,E1 -25827.814,E2 -25827.814} C_VEL
LIN {X 0,Y 190.385,Z 539.589,A -85,B 0,C 180,E1 -25830,E2 -25830} C_VEL
LIN {X 0,Y 182.922,Z 539.534,A -85,B 0,C 180,E1 -25832.669,E2 -25832.669} C_VEL
LIN {X 0,Y 176.425,Z 539.06,A -85,B 0,C 180,E1 -25835.214,E2 -25835.214} C_VEL
LIN {X 0,Y 166.564,Z 537.194,A -85,B 0,C 180,E1 -25839.717,E2 -25839.717} C_VEL
LIN {X 0,Y 159.259,Z 534.708,A -85,B 0,C 180,E1 -25843.875,E2 -25843.875} C_VEL
LIN {X 0,Y 154.51,Z 532.294,A -85,B 0,C 180,E1 -25847.22,E2 -25847.22} C_VEL
LIN {X 0,Y 149.215,Z 527.882,A -85,B 0,C 180,E1 -25852.136,E2 -25852.136} C_VEL
LIN {X 0,Y 145.464,Z 522.161,A -85,B 0,C 180,E1 -25857.322,E2 -25857.322} C_VEL
LIN {X 0,Y 143.527,Z 516.309,A -85,B 0,C 180,E1 -25861.762,E2 -25861.762} C_VEL
LIN {X 0,Y 142.802,Z 510.79,A -85,B 0,C 180,E1 -25865.334,E2 -25865.334} C_VEL
LIN {X 0,Y 142.52,Z 503.916,A -85,B 0,C 180,E1 -25869.173,E2 -25869.173} C_VEL
LIN {X 0,Y 141.464,Z 495.579,A -85,B 0,C 180,E1 -25873.617,E2 -25873.617} C_VEL
LIN {X 0,Y 140.039,Z 488.639,A -85,B 0,C 180,E1 -25877.353,E2 -25877.353} C_VEL
LIN {X 0,Y 137.41,Z 480.353,A -85,B 0,C 180,E1 -25882.141,E2 -25882.141} C_VEL
LIN {X 0,Y 134.495,Z 473.323,A -85,B 0,C 180,E1 -25886.728,E2 -25886.728} C_VEL
LIN {X 0,Y 132.521,Z 469.064,A -85,B 0,C 180,E1 -25889.749,E2 -25889.749} C_VEL
LIN {X 0,Y 129.609,Z 464.088,A -85,B 0,C 180,E1 -25894.293,E2 -25894.293} C_VEL
LIN {X 0,Y 126.929,Z 459.744,A -85,B 0,C 180,E1 -25898.908,E2 -25898.908} C_VEL
LIN {X 0,Y 125.014,Z 456.931,A -85,B 0,C 180,E1 -25902.881,E2 -25902.881} C_VEL
LIN {X 0,Y 124.79,Z 456.202,A -85,B 0,C 180,E1 -25903.647,E2 -25903.647} C_VEL
LIN {X 0,Y 122.988,Z 454.116,A -85,B 0,C 180,E1 -25908.465,E2 -25908.465} C_VEL
LIN {X 0,Y 121.573,Z 450.629,A -85,B 0,C 180,E1 -25920.209,E2 -25920.209} C_VEL
LIN {X 0,Y 124.63,Z 455.619,A -85,B 0,C 180,E1 -25934.702,E2 -25934.702} C_VEL
LIN {X 0,Y 126.426,Z 460.134,A -85,B 0,C 180,E1 -25939.486,E2 -25939.486} C_VEL
LIN {X 0,Y 127.305,Z 461.293,A -85,B 0,C 180,E1 -25941.031,E2 -25941.031} C_VEL
LIN {X 0,Y 130.238,Z 467.127,A -85,B 0,C 180,E1 -25946.138,E2 -25946.138} C_VEL
LIN {X 0,Y 131.577,Z 470.878,A -85,B 0,C 180,E1 -25948.735,E2 -25948.735} C_VEL
LIN {X 0,Y 132.491,Z 473.128,A -85,B 0,C 180,E1 -25950.262,E2 -25950.262} C_VEL
LIN {X 0,Y 134.178,Z 477.697,A -85,B 0,C 180,E1 -25953.065,E2 -25953.065} C_VEL
LIN {X 0,Y 136.061,Z 484.925,A -85,B 0,C 180,E1 -25956.982,E2 -25956.982} C_VEL
LIN {X 0,Y 136.583,Z 490.339,A -85,B 0,C 180,E1 -25959.481,E2 -25959.481} C_VEL
LIN {X 0,Y 136.429,Z 497.718,A -85,B 0,C 180,E1 -25962.599,E2 -25962.599} C_VEL
LIN {X 0,Y 135.407,Z 506,A -85,B 0,C 180,E1 -25966.154,E2 -25966.154} C_VEL
LIN {X 0,Y 134.065,Z 512.417,A -85,B 0,C 180,E1 -25969.059,E2 -25969.059} C_VEL
LIN {X 0,Y 132.532,Z 517.351,A -85,B 0,C 180,E1 -25971.458,E2 -25971.458} C_VEL
LIN {X 0,Y 127.381,Z 525.685,A -85,B 0,C 180,E1 -25975.561,E2 -25975.561} C_VEL
LIN {X 0,Y 123.68,Z 531.35,A -85,B 0,C 180,E1 -25979.242,E2 -25979.242} C_VEL
LIN {X 0,Y 119.651,Z 536.843,A -85,B 0,C 180,E1 -25983.862,E2 -25983.862} C_VEL
LIN {X 0,Y 116.424,Z 541.171,A -85,B 0,C 180,E1 -25988.765,E2 -25988.765} C_VEL
LIN {X 0,Y 114.856,Z 543.545,A -85,B 0,C 180,E1 -25992.184,E2 -25992.184} C_VEL
LIN {X 0,Y 113.66,Z 545.352,A -85,B 0,C 180,E1 -25995.68,E2 -25995.68} C_VEL
LIN {X 0,Y 112.343,Z 547.816,A -85,B 0,C 180,E1 -26002.812,E2 -26002.812} C_VEL
LIN {X 0,Y 112.14,Z 548.413,A -85,B 0,C 180,E1 -26006.406,E2 -26006.406} C_VEL
LIN {X 0,Y 112.252,Z 548.575,A -85,B 0,C 180,E1 -26009.999,E2 -26009.999} C_VEL
LIN {X 0,Y 112.14,Z 548.413,A -85,B 0,C 180,E1 -26013.592,E2 -26013.592} C_VEL
LIN {X 0,Y 112.342,Z 547.817,A -85,B 0,C 180,E1 -26017.187,E2 -26017.187} C_VEL
LIN {X 0,Y 113.66,Z 545.353,A -85,B 0,C 180,E1 -26024.319,E2 -26024.319} C_VEL
LIN {X 0,Y 115.574,Z 542.392,A -85,B 0,C 180,E1 -26029.538,E2 -26029.538} C_VEL
LIN {X 0,Y 118.484,Z 538.399,A -85,B 0,C 180,E1 -26034.531,E2 -26034.531} C_VEL
LIN {X 0,Y 122.208,Z 533.266,A -85,B 0,C 180,E1 -26039.262,E2 -26039.262} C_VEL
LIN {X 0,Y 126.161,Z 527.488,A -85,B 0,C 180,E1 -26043.319,E2 -26043.319} C_VEL
LIN {X 0,Y 129.873,Z 521.679,A -85,B 0,C 180,E1 -26046.53,E2 -26046.53} C_VEL
LIN {X 0,Y 132.533,Z 517.354,A -85,B 0,C 180,E1 -26048.54,E2 -26048.54} C_VEL
LIN {X 0,Y 134.542,Z 510.648,A -85,B 0,C 180,E1 -26051.759,E2 -26051.759} C_VEL
LIN {X 0,Y 135.892,Z 502.703,A -85,B 0,C 180,E1 -26055.323,E2 -26055.323} C_VEL
LIN {X 0,Y 136.562,Z 494.907,A -85,B 0,C 180,E1 -26058.642,E2 -26058.642} C_VEL
LIN {X 0,Y 136.423,Z 487.487,A -85,B 0,C 180,E1 -26061.814,E2 -26061.814} C_VEL
LIN {X 0,Y 135.589,Z 482.847,A -85,B 0,C 180,E1 -26064.058,E2 -26064.058} C_VEL
LIN {X 0,Y 133.456,Z 475.492,A -85,B 0,C 180,E1 -26068.221,E2 -26068.221} C_VEL
LIN {X 0,Y 131.584,Z 470.859,A -85,B 0,C 180,E1 -26071.267,E2 -26071.267} C_VEL
LIN {X 0,Y 129.908,Z 466.601,A -85,B 0,C 180,E1 -26074.353,E2 -26074.353} C_VEL
LIN {X 0,Y 127.306,Z 461.288,A -85,B 0,C 180,E1 -26078.969,E2 -26078.969} C_VEL
LIN {X 0,Y 125.843,Z 459.212,A -85,B 0,C 180,E1 -26081.691,E2 -26081.691} C_VEL
LIN {X 0,Y 124.641,Z 455.575,A -85,B 0,C 180,E1 -26085.299,E2 -26085.299} C_VEL
LIN {X 0,Y 121.576,Z 450.603,A -85,B 0,C 180,E1 -26099.998,E2 -26099.998} C_VEL
LIN {X 0,Y 123.559,Z 454.66,A -85,B 0,C 180,E1 -26113.149,E2 -26113.149} C_VEL
LIN {X 0,Y 124.796,Z 456.184,A -85,B 0,C 180,E1 -26116.353,E2 -26116.353} C_VEL
LIN {X 0,Y 127.65,Z 460.847,A -85,B 0,C 180,E1 -26122.401,E2 -26122.401} C_VEL
LIN {X 0,Y 128.801,Z 463.541,A -85,B 0,C 180,E1 -26124.688,E2 -26124.688} C_VEL
LIN {X 0,Y 129.335,Z 467.146,A -85,B 0,C 180,E1 -26126.78,E2 -26126.78} C_VEL
LIN {X 0,Y 130.052,Z 477.789,A -85,B 0,C 180,E1 -26132.133,E2 -26132.133} C_VEL
LIN {X 0,Y 130.669,Z 480.023,A -85,B 0,C 180,E1 -26133.583,E2 -26133.583} C_VEL
LIN {X 0,Y 133.017,Z 486.806,A -85,B 0,C 180,E1 -26138.264,E2 -26138.264} C_VEL
LIN {X 0,Y 134.511,Z 492.631,A -85,B 0,C 180,E1 -26141.868,E2 -26141.868} C_VEL
LIN {X 0,Y 135.577,Z 498.802,A -85,B 0,C 180,E1 -26145.457,E2 -26145.457} C_VEL
LIN {X 0,Y 136.219,Z 506.145,A -85,B 0,C 180,E1 -26149.743,E2 -26149.743} C_VEL
LIN {X 0,Y 136.346,Z 513.898,A -85,B 0,C 180,E1 -26154.559,E2 -26154.559} C_VEL
LIN {X 0,Y 137.272,Z 520.201,A -85,B 0,C 180,E1 -26159.206,E2 -26159.206} C_VEL
LIN {X 0,Y 138.78,Z 524.512,A -85,B 0,C 180,E1 -26162.887,E2 -26162.887} C_VEL
LIN {X 0,Y 142.191,Z 529.44,A -85,B 0,C 180,E1 -26167.961,E2 -26167.961} C_VEL
LIN {X 0,Y 147.07,Z 533.374,A -85,B 0,C 180,E1 -26172.883,E2 -26172.883} C_VEL
LIN {X 0,Y 152.179,Z 535.885,A -85,B 0,C 180,E1 -26176.65,E2 -26176.65} C_VEL
LIN {X 0,Y 157.141,Z 537.482,A -85,B 0,C 180,E1 -26179.707,E2 -26179.707} C_VEL
LIN {X 0,Y 169.18,Z 539.561,A -85,B 0,C 180,E1 -26185.54,E2 -26185.54} C_VEL
LIN {X 0,Y 175.786,Z 539.963,A -85,B 0,C 180,E1 -26188.161,E2 -26188.161} C_VEL
LIN {X 0,Y 180.862,Z 539.867,A -85,B 0,C 180,E1 -26190,E2 -26190} C_VEL
LIN {X 0,Y 174.579,Z 539.9,A -85,B 0,C 180,E1 -26192.308,E2 -26192.308} C_VEL
LIN {X 0,Y 168.455,Z 539.51,A -85,B 0,C 180,E1 -26194.787,E2 -26194.787} C_VEL
LIN {X 0,Y 157.117,Z 537.474,A -85,B 0,C 180,E1 -26200.307,E2 -26200.307} C_VEL
LIN {X 0,Y 149.855,Z 534.841,A -85,B 0,C 180,E1 -26204.947,E2 -26204.947} C_VEL
LIN {X 0,Y 145.694,Z 532.518,A -85,B 0,C 180,E1 -26208.354,E2 -26208.354} C_VEL
LIN {X 0,Y 141.037,Z 528.146,A -85,B 0,C 180,E1 -26213.494,E2 -26213.494} C_VEL
LIN {X 0,Y 138.127,Z 523.056,A -85,B 0,C 180,E1 -26218.426,E2 -26218.426} C_VEL
LIN {X 0,Y 136.492,Z 516.317,A -85,B 0,C 180,E1 -26223.769,E2 -26223.769} C_VEL
LIN {X 0,Y 136.239,Z 509.46,A -85,B 0,C 180,E1 -26228.245,E2 -26228.245} C_VEL
LIN {X 0,Y 136.143,Z 504.515,A -85,B 0,C 180,E1 -26231.21,E2 -26231.21} C_VEL
LIN {X 0,Y 135.35,Z 497.156,A -85,B 0,C 180,E1 -26235.499,E2 -26235.499} C_VEL
LIN {X 0,Y 133.837,Z 489.871,A -85,B 0,C 180,E1 -26239.885,E2 -26239.885} C_VEL
LIN {X 0,Y 131.845,Z 483.329,A -85,B 0,C 180,E1 -26244.103,E2 -26244.103} C_VEL
LIN {X 0,Y 129.27,Z 476.781,A -85,B 0,C 180,E1 -26248.905,E2 -26248.905} C_VEL
LIN {X 0,Y 127.982,Z 473.7,A -85,B 0,C 180,E1 -26251.476,E2 -26251.476} C_VEL
LIN {X 0,Y 125.907,Z 469.783,A -85,B 0,C 180,E1 -26255.253,E2 -26255.253} C_VEL
LIN {X 0,Y 124.408,Z 466.846,A -85,B 0,C 180,E1 -26258.459,E2 -26258.459} C_VEL
LIN {X 0,Y 122.4,Z 463.496,A -85,B 0,C 180,E1 -26263.318,E2 -26263.318} C_VEL
LIN {X 0,Y 121.295,Z 461.53,A -85,B 0,C 180,E1 -26266.601,E2 -26266.601} C_VEL
LIN {X 0,Y 119.639,Z 457.549,A -85,B 0,C 180,E1 -26280.002,E2 -26280.002} C_VEL
LIN {X 0,Y 121.751,Z 461.837,A -85,B 0,C 180,E1 -26293.352,E2 -26293.352} C_VEL
LIN {X 0,Y 124.753,Z 468.723,A -85,B 0,C 180,E1 -26301.482,E2 -26301.482} C_VEL
LIN {X 0,Y 126.56,Z 473.216,A -85,B 0,C 180,E1 -26305.493,E2 -26305.493} C_VEL
LIN {X 0,Y 128.394,Z 478.732,A -85,B 0,C 180,E1 -26309.516,E2 -26309.516} C_VEL
LIN {X 0,Y 129.984,Z 484.322,A -85,B 0,C 180,E1 -26313.14,E2 -26313.14} C_VEL
LIN {X 0,Y 131.017,Z 490.07,A -85,B 0,C 180,E1 -26316.426,E2 -26316.426} C_VEL
LIN {X 0,Y 131.056,Z 495.702,A -85,B 0,C 180,E1 -26319.059,E2 -26319.059} C_VEL
LIN {X 0,Y 130.385,Z 502.461,A -85,B 0,C 180,E1 -26322.172,E2 -26322.172} C_VEL
LIN {X 0,Y 128.684,Z 511.181,A -85,B 0,C 180,E1 -26326.31,E2 -26326.31} C_VEL
LIN {X 0,Y 126.861,Z 517.132,A -85,B 0,C 180,E1 -26329.387,E2 -26329.387} C_VEL
LIN {X 0,Y 124.225,Z 521.465,A -85,B 0,C 180,E1 -26331.514,E2 -26331.514} C_VEL
LIN {X 0,Y 119.912,Z 527.778,A -85,B 0,C 180,E1 -26335.141,E2 -26335.141} C_VEL
LIN {X 0,Y 116.064,Z 533.053,A -85,B 0,C 180,E1 -26339.022,E2 -26339.022} C_VEL
LIN {X 0,Y 112.05,Z 538.186,A -85,B 0,C 180,E1 -26343.956,E2 -26343.956} C_VEL
LIN {X 0,Y 108.881,Z 542.179,A -85,B 0,C 180,E1 -26349.205,E2 -26349.205} C_VEL
LIN {X 0,Y 106.767,Z 545.14,A -85,B 0,C 180,E1 -26354.733,E2 -26354.733} C_VEL
LIN {X 0,Y 105.285,Z 547.605,A -85,B 0,C 180,E1 -26362.327,E2 -26362.327} C_VEL
LIN {X 0,Y 105.049,Z 548.202,A -85,B 0,C 180,E1 -26366.163,E2 -26366.163} C_VEL
LIN {X 0,Y 105.171,Z 548.365,A -85,B 0,C 180,E1 -26369.999,E2 -26369.999} C_VEL
LIN {X 0,Y 105.049,Z 548.202,A -85,B 0,C 180,E1 -26373.835,E2 -26373.835} C_VEL
LIN {X 0,Y 105.285,Z 547.605,A -85,B 0,C 180,E1 -26377.671,E2 -26377.671} C_VEL
LIN {X 0,Y 106.766,Z 545.141,A -85,B 0,C 180,E1 -26385.265,E2 -26385.265} C_VEL
LIN {X 0,Y 108.879,Z 542.18,A -85,B 0,C 180,E1 -26390.793,E2 -26390.793} C_VEL
LIN {X 0,Y 112.047,Z 538.187,A -85,B 0,C 180,E1 -26396.043,E2 -26396.043} C_VEL
LIN {X 0,Y 116.055,Z 533.054,A -85,B 0,C 180,E1 -26400.979,E2 -26400.979} C_VEL
LIN {X 0,Y 119.807,Z 527.898,A -85,B 0,C 180,E1 -26404.787,E2 -26404.787} C_VEL
LIN {X 0,Y 124.223,Z 521.468,A -85,B 0,C 180,E1 -26408.485,E2 -26408.485} C_VEL
LIN {X 0,Y 126.107,Z 518.707,A -85,B 0,C 180,E1 -26409.857,E2 -26409.857} C_VEL
LIN {X 0,Y 127.407,Z 515.49,A -85,B 0,C 180,E1 -26411.447,E2 -26411.447} C_VEL
LIN {X 0,Y 128.977,Z 509.982,A -85,B 0,C 180,E1 -26414.249,E2 -26414.249} C_VEL
LIN {X 0,Y 130.347,Z 502.463,A -85,B 0,C 180,E1 -26417.845,E2 -26417.845} C_VEL
LIN {X 0,Y 131.122,Z 494.574,A -85,B 0,C 180,E1 -26421.457,E2 -26421.457} C_VEL
LIN {X 0,Y 130.958,Z 489.623,A -85,B 0,C 180,E1 -26423.818,E2 -26423.818} C_VEL
LIN {X 0,Y 129.852,Z 483.657,A -85,B 0,C 180,E1 -26427.231,E2 -26427.231} C_VEL
LIN {X 0,Y 128.061,Z 477.348,A -85,B 0,C 180,E1 -26431.409,E2 -26431.409} C_VEL
LIN {X 0,Y 126.178,Z 472.245,A -85,B 0,C 180,E1 -26435.306,E2 -26435.306} C_VEL
LIN {X 0,Y 124.087,Z 467.207,A -85,B 0,C 180,E1 -26440.132,E2 -26440.132} C_VEL
LIN {X 0,Y 121.752,Z 461.832,A -85,B 0,C 180,E1 -26446.648,E2 -26446.648} C_VEL
LIN {X 0,Y 119.637,Z 457.555,A -85,B 0,C 180,E1 -26459.998,E2 -26459.998} C_VEL
LIN {X 0,Y 121.293,Z 461.535,A -85,B 0,C 180,E1 -26473.399,E2 -26473.399} C_VEL
LIN {X 0,Y 123.665,Z 465.724,A -85,B 0,C 180,E1 -26479.935,E2 -26479.935} C_VEL
LIN {X 0,Y 124.404,Z 466.856,A -85,B 0,C 180,E1 -26481.541,E2 -26481.541} C_VEL
LIN {X 0,Y 126.798,Z 471.259,A -85,B 0,C 180,E1 -26486.32,E2 -26486.32} C_VEL
LIN {X 0,Y 128.867,Z 475.769,A -85,B 0,C 180,E1 -26490.294,E2 -26490.294} C_VEL
LIN {X 0,Y 130.669,Z 480.023,A -85,B 0,C 180,E1 -26493.583,E2 -26493.583} C_VEL
LIN {X 0,Y 131.279,Z 482.229,A -85,B 0,C 180,E1 -26494.985,E2 -26494.985} C_VEL
LIN {X 0,Y 131.461,Z 486.109,A -85,B 0,C 180,E1 -26496.94,E2 -26496.94} C_VEL
LIN {X 0,Y 131.012,Z 490.308,A -85,B 0,C 180,E1 -26498.78,E2 -26498.78} C_VEL
LIN {X 0,Y 129.544,Z 499.387,A -85,B 0,C 180,E1 -26502.957,E2 -26502.957} C_VEL
LIN {X 0,Y 129.528,Z 501.146,A -85,B 0,C 180,E1 -26504.031,E2 -26504.031} C_VEL
LIN {X 0,Y 129.853,Z 506.563,A -85,B 0,C 180,E1 -26507.431,E2 -26507.431} C_VEL
LIN {X 0,Y 129.853,Z 512.801,A -85,B 0,C 180,E1 -26511.509,E2 -26511.509} C_VEL
LIN {X 0,Y 130.158,Z 520.45,A -85,B 0,C 180,E1 -26517.32,E2 -26517.32} C_VEL
LIN {X 0,Y 131.205,Z 524.767,A -85,B 0,C 180,E1 -26521.18,E2 -26521.18} C_VEL
LIN {X 0,Y 134.275,Z 529.972,A -85,B 0,C 180,E1 -26526.888,E2 -26526.888} C_VEL
LIN {X 0,Y 138.961,Z 534.001,A -85,B 0,C 180,E1 -26532.336,E2 -26532.336} C_VEL
LIN {X 0,Y 144.386,Z 536.643,A -85,B 0,C 180,E1 -26536.773,E2 -26536.773} C_VEL
LIN {X 0,Y 149.755,Z 538.327,A -85,B 0,C 180,E1 -26540.231,E2 -26540.231} C_VEL
LIN {X 0,Y 158.795,Z 539.794,A -85,B 0,C 180,E1 -26544.922,E2 -26544.922} C_VEL
LIN {X 0,Y 168.691,Z 540.223,A -85,B 0,C 180,E1 -26549.047,E2 -26549.047} C_VEL
LIN {X 0,Y 171.24,Z 540.148,A -85,B 0,C 180,E1 -26550.001,E2 -26550.001} C_VEL
LIN {X 0,Y 161.972,Z 539.998,A -85,B 0,C 180,E1 -26553.672,E2 -26553.672} C_VEL
LIN {X 0,Y 153.032,Z 538.939,A -85,B 0,C 180,E1 -26557.92,E2 -26557.92} C_VEL
LIN {X 0,Y 147.759,Z 537.757,A -85,B 0,C 180,E1 -26560.968,E2 -26560.968} C_VEL
LIN {X 0,Y 143.04,Z 536.164,A -85,B 0,C 180,E1 -26564.222,E2 -26564.222} C_VEL
LIN {X 0,Y 137.316,Z 532.88,A -85,B 0,C 180,E1 -26569.403,E2 -26569.403} C_VEL
LIN {X 0,Y 132.635,Z 527.691,A -85,B 0,C 180,E1 -26575.742,E2 -26575.742} C_VEL
LIN {X 0,Y 130.646,Z 522.823,A -85,B 0,C 180,E1 -26580.608,E2 -26580.608} C_VEL
LIN {X 0,Y 129.756,Z 516.72,A -85,B 0,C 180,E1 -26585.668,E2 -26585.668} C_VEL
LIN {X 0,Y 129.909,Z 510.651,A -85,B 0,C 180,E1 -26589.872,E2 -26589.872} C_VEL
LIN {X 0,Y 129.787,Z 504.684,A -85,B 0,C 180,E1 -26593.767,E2 -26593.767} C_VEL
LIN {X 0,Y 129.201,Z 498.56,A -85,B 0,C 180,E1 -26597.71,E2 -26597.71} C_VEL
LIN {X 0,Y 127.963,Z 492.109,A -85,B 0,C 180,E1 -26601.994,E2 -26601.994} C_VEL
LIN {X 0,Y 126.14,Z 485.693,A -85,B 0,C 180,E1 -26606.693,E2 -26606.693} C_VEL
LIN {X 0,Y 124.12,Z 479.807,A -85,B 0,C 180,E1 -26611.606,E2 -26611.606} C_VEL
LIN {X 0,Y 122.071,Z 475.404,A -85,B 0,C 180,E1 -26616.236,E2 -26616.236} C_VEL
LIN {X 0,Y 120.836,Z 472.623,A -85,B 0,C 180,E1 -26619.578,E2 -26619.578} C_VEL
LIN {X 0,Y 118.638,Z 468.418,A -85,B 0,C 180,E1 -26626.295,E2 -26626.295} C_VEL
LIN {X 0,Y 117.263,Z 466.187,A -85,B 0,C 180,E1 -26633.118,E2 -26633.118} C_VEL
LIN {X 0,Y 117.316,Z 464.349,A -85,B 0,C 180,E1 -26640.002,E2 -26640.002} C_VEL
LIN {X 0,Y 118.221,Z 467.446,A -85,B 0,C 180,E1 -26650.275,E2 -26650.275} C_VEL
LIN {X 0,Y 119.138,Z 468.918,A -85,B 0,C 180,E1 -26653.65,E2 -26653.65} C_VEL
LIN {X 0,Y 121.146,Z 474.383,A -85,B 0,C 180,E1 -26660.372,E2 -26660.372} C_VEL
LIN {X 0,Y 122.599,Z 478.78,A -85,B 0,C 180,E1 -26664.559,E2 -26664.559} C_VEL
LIN {X 0,Y 124.374,Z 485.164,A -85,B 0,C 180,E1 -26669.521,E2 -26669.521} C_VEL
LIN {X 0,Y 125.326,Z 490.364,A -85,B 0,C 180,E1 -26673.052,E2 -26673.052} C_VEL
LIN {X 0,Y 125.754,Z 495.456,A -85,B 0,C 180,E1 -26675.985,E2 -26675.985} C_VEL
LIN {X 0,Y 124.87,Z 503.437,A -85,B 0,C 180,E1 -26679.995,E2 -26679.995} C_VEL
LIN {X 0,Y 122.666,Z 512.607,A -85,B 0,C 180,E1 -26684.719,E2 -26684.719} C_VEL
LIN {X 0,Y 120.624,Z 518.489,A -85,B 0,C 180,E1 -26687.93,E2 -26687.93} C_VEL
LIN {X 0,Y 114.997,Z 526.417,A -85,B 0,C 180,E1 -26692.327,E2 -26692.327} C_VEL
LIN {X 0,Y 110.026,Z 532.841,A -85,B 0,C 180,E1 -26697.115,E2 -26697.115} C_VEL
LIN {X 0,Y 105.701,Z 537.974,A -85,B 0,C 180,E1 -26702.262,E2 -26702.262} C_VEL
LIN {X 0,Y 102.253,Z 541.967,A -85,B 0,C 180,E1 -26707.788,E2 -26707.788} C_VEL
LIN {X 0,Y 99.891,Z 544.927,A -85,B 0,C 180,E1 -26713.654,E2 -26713.654} C_VEL
LIN {X 0,Y 98.253,Z 547.393,A -85,B 0,C 180,E1 -26721.774,E2 -26721.774} C_VEL
LIN {X 0,Y 97.955,Z 547.99,A -85,B 0,C 180,E1 -26725.885,E2 -26725.885} C_VEL
LIN {X 0,Y 98.077,Z 548.154,A -85,B 0,C 180,E1 -26729.999,E2 -26729.999} C_VEL
LIN {X 0,Y 97.955,Z 547.99,A -85,B 0,C 180,E1 -26734.113,E2 -26734.113} C_VEL
LIN {X 0,Y 98.253,Z 547.393,A -85,B 0,C 180,E1 -26738.224,E2 -26738.224} C_VEL
LIN {X 0,Y 99.891,Z 544.928,A -85,B 0,C 180,E1 -26746.344,E2 -26746.344} C_VEL
LIN {X 0,Y 102.252,Z 541.968,A -85,B 0,C 180,E1 -26752.21,E2 -26752.21} C_VEL
LIN {X 0,Y 105.698,Z 537.975,A -85,B 0,C 180,E1 -26757.737,E2 -26757.737} C_VEL
LIN {X 0,Y 110.017,Z 532.843,A -85,B 0,C 180,E1 -26762.886,E2 -26762.886} C_VEL
LIN {X 0,Y 114.995,Z 526.419,A -85,B 0,C 180,E1 -26767.671,E2 -26767.671} C_VEL
LIN {X 0,Y 120.604,Z 518.49,A -85,B 0,C 180,E1 -26772.076,E2 -26772.076} C_VEL
LIN {X 0,Y 123.12,Z 511.147,A -85,B 0,C 180,E1 -26776.087,E2 -26776.087} C_VEL
LIN {X 0,Y 125.022,Z 502.194,A -85,B 0,C 180,E1 -26780.63,E2 -26780.63} C_VEL
LIN {X 0,Y 125.755,Z 495.46,A -85,B 0,C 180,E1 -26784.012,E2 -26784.012} C_VEL
LIN {X 0,Y 125.325,Z 490.366,A -85,B 0,C 180,E1 -26786.948,E2 -26786.948} C_VEL
LIN {X 0,Y 124.373,Z 485.165,A -85,B 0,C 180,E1 -26790.479,E2 -26790.479} C_VEL
LIN {X 0,Y 122.328,Z 477.819,A -85,B 0,C 180,E1 -26796.285,E2 -26796.285} C_VEL
LIN {X 0,Y 121.149,Z 474.373,A -85,B 0,C 180,E1 -26799.629,E2 -26799.629} C_VEL
LIN {X 0,Y 119.135,Z 468.926,A -85,B 0,C 180,E1 -26806.349,E2 -26806.349} C_VEL
LIN {X 0,Y 118.22,Z 467.448,A -85,B 0,C 180,E1 -26809.725,E2 -26809.725} C_VEL
LIN {X 0,Y 117.318,Z 464.343,A -85,B 0,C 180,E1 -26819.998,E2 -26819.998} C_VEL
LIN {X 0,Y 117.809,Z 467.146,A -85,B 0,C 180,E1 -26830.308,E2 -26830.308} C_VEL
LIN {X 0,Y 118.639,Z 468.415,A -85,B 0,C 180,E1 -26833.705,E2 -26833.705} C_VEL
LIN {X 0,Y 120.838,Z 472.618,A -85,B 0,C 180,E1 -26840.422,E2 -26840.422} C_VEL
LIN {X 0,Y 122.797,Z 476.8,A -85,B 0,C 180,E1 -26845.417,E2 -26845.417} C_VEL
LIN {X 0,Y 124.538,Z 480.998,A -85,B 0,C 180,E1 -26849.388,E2 -26849.388} C_VEL
LIN {X 0,Y 126.723,Z 487.391,A -85,B 0,C 180,E1 -26854.641,E2 -26854.641} C_VEL
LIN {X 0,Y 127.899,Z 491.539,A -85,B 0,C 180,E1 -26857.634,E2 -26857.634} C_VEL
LIN {X 0,Y 129.217,Z 498.548,A -85,B 0,C 180,E1 -26862.291,E2 -26862.291} C_VEL
LIN {X 0,Y 129.528,Z 501.146,A -85,B 0,C 180,E1 -26864.031,E2 -26864.031} C_VEL
LIN {X 0,Y 129.088,Z 504.961,A -85,B 0,C 180,E1 -26866.08,E2 -26866.08} C_VEL
LIN {X 0,Y 127.711,Z 508.861,A -85,B 0,C 180,E1 -26867.998,E2 -26867.998} C_VEL
LIN {X 0,Y 123.853,Z 517.439,A -85,B 0,C 180,E1 -26872.69,E2 -26872.69} C_VEL
LIN {X 0,Y 123.276,Z 520.462,A -85,B 0,C 180,E1 -26875.038,E2 -26875.038} C_VEL
LIN {X 0,Y 123.91,Z 525.017,A -85,B 0,C 180,E1 -26879.306,E2 -26879.306} C_VEL
LIN {X 0,Y 126.319,Z 530.362,A -85,B 0,C 180,E1 -26885.492,E2 -26885.492} C_VEL
LIN {X 0,Y 130.426,Z 534.269,A -85,B 0,C 180,E1 -26891.138,E2 -26891.138} C_VEL
LIN {X 0,Y 134.082,Z 536.441,A -85,B 0,C 180,E1 -26894.807,E2 -26894.807} C_VEL
LIN {X 0,Y 142.377,Z 538.997,A -85,B 0,C 180,E1 -26900.826,E2 -26900.826} C_VEL
LIN {X 0,Y 149.171,Z 540.079,A -85,B 0,C 180,E1 -26904.594,E2 -26904.594} C_VEL
LIN {X 0,Y 155.224,Z 540.468,A -85,B 0,C 180,E1 -26907.406,E2 -26907.406} C_VEL
LIN {X 0,Y 161.588,Z 540.43,A -85,B 0,C 180,E1 -26910.001,E2 -26910.001} C_VEL
LIN {X 0,Y 154.796,Z 540.437,A -85,B 0,C 180,E1 -26912.797,E2 -26912.797} C_VEL
LIN {X 0,Y 148.349,Z 540.018,A -85,B 0,C 180,E1 -26915.823,E2 -26915.823} C_VEL
LIN {X 0,Y 138.497,Z 538.039,A -85,B 0,C 180,E1 -26921.712,E2 -26921.712} C_VEL
LIN {X 0,Y 132.217,Z 535.452,A -85,B 0,C 180,E1 -26926.911,E2 -26926.911} C_VEL
LIN {X 0,Y 127.404,Z 531.692,A -85,B 0,C 180,E1 -26932.715,E2 -26932.715} C_VEL
LIN {X 0,Y 125.28,Z 528.664,A -85,B 0,C 180,E1 -26936.666,E2 -26936.666} C_VEL
LIN {X 0,Y 123.453,Z 522.808,A -85,B 0,C 180,E1 -26942.834,E2 -26942.834} C_VEL
LIN {X 0,Y 123.233,Z 518.064,A -85,B 0,C 180,E1 -26947.023,E2 -26947.023} C_VEL
LIN {X 0,Y 123.669,Z 510.835,A -85,B 0,C 180,E1 -26952.375,E2 -26952.375} C_VEL
LIN {X 0,Y 123.581,Z 504.355,A -85,B 0,C 180,E1 -26956.968,E2 -26956.968} C_VEL
LIN {X 0,Y 123,Z 498.737,A -85,B 0,C 180,E1 -26961.061,E2 -26961.061} C_VEL
LIN {X 0,Y 121.875,Z 493.101,A -85,B 0,C 180,E1 -26965.365,E2 -26965.365} C_VEL
LIN {X 0,Y 120.623,Z 488.451,A -85,B 0,C 180,E1 -26969.352,E2 -26969.352} C_VEL
LIN {X 0,Y 119.215,Z 483.865,A -85,B 0,C 180,E1 -26973.762,E2 -26973.762} C_VEL
LIN {X 0,Y 117.437,Z 479.533,A -85,B 0,C 180,E1 -26978.959,E2 -26978.959} C_VEL
LIN {X 0,Y 115.999,Z 476.141,A -85,B 0,C 180,E1 -26984.181,E2 -26984.181} C_VEL
LIN {X 0,Y 115.515,Z 474.732,A -85,B 0,C 180,E1 -26986.767,E2 -26986.767} C_VEL
LIN {X 0,Y 114.413,Z 472.76,A -85,B 0,C 180,E1 -26992.945,E2 -26992.945} C_VEL
LIN {X 0,Y 114.517,Z 470.957,A -85,B 0,C 180,E1 -27000.002,E2 -27000.002} C_VEL
LIN {X 0,Y 115.364,Z 474.095,A -85,B 0,C 180,E1 -27010.533,E2 -27010.533} C_VEL
LIN {X 0,Y 116.148,Z 476.384,A -85,B 0,C 180,E1 -27014.501,E2 -27014.501} C_VEL
LIN {X 0,Y 117.277,Z 479.87,A -85,B 0,C 180,E1 -27019.246,E2 -27019.246} C_VEL
LIN {X 0,Y 118.394,Z 483.986,A -85,B 0,C 180,E1 -27023.424,E2 -27023.424} C_VEL
LIN {X 0,Y 119.68,Z 490.436,A -85,B 0,C 180,E1 -27028.883,E2 -27028.883} C_VEL
LIN {X 0,Y 120.351,Z 496.026,A -85,B 0,C 180,E1 -27032.842,E2 -27032.842} C_VEL
LIN {X 0,Y 120.192,Z 499.645,A -85,B 0,C 180,E1 -27035.053,E2 -27035.053} C_VEL
LIN {X 0,Y 119.276,Z 505.044,A -85,B 0,C 180,E1 -27037.982,E2 -27037.982} C_VEL
LIN {X 0,Y 117.374,Z 512.12,A -85,B 0,C 180,E1 -27041.85,E2 -27041.85} C_VEL
LIN {X 0,Y 115.144,Z 518.264,A -85,B 0,C 180,E1 -27045.418,E2 -27045.418} C_VEL
LIN {X 0,Y 114.426,Z 519.663,A -85,B 0,C 180,E1 -27046.293,E2 -27046.293} C_VEL
LIN {X 0,Y 109.446,Z 526.205,A -85,B 0,C 180,E1 -27050.048,E2 -27050.048} C_VEL
LIN {X 0,Y 105.808,Z 530.711,A -85,B 0,C 180,E1 -27053.287,E2 -27053.287} C_VEL
LIN {X 0,Y 100.852,Z 536.205,A -85,B 0,C 180,E1 -27058.49,E2 -27058.49} C_VEL
LIN {X 0,Y 96.834,Z 540.536,A -85,B 0,C 180,E1 -27064.184,E2 -27064.184} C_VEL
LIN {X 0,Y 94.672,Z 542.907,A -85,B 0,C 180,E1 -27068.211,E2 -27068.211} C_VEL
LIN {X 0,Y 93.063,Z 544.715,A -85,B 0,C 180,E1 -27072.417,E2 -27072.417} C_VEL
LIN {X 0,Y 91.2,Z 547.181,A -85,B 0,C 180,E1 -27081.133,E2 -27081.133} C_VEL
LIN {X 0,Y 90.885,Z 547.779,A -85,B 0,C 180,E1 -27085.564,E2 -27085.564} C_VEL
LIN {X 0,Y 90.976,Z 547.942,A -85,B 0,C 180,E1 -27089.999,E2 -27089.999} C_VEL
LIN {X 0,Y 90.885,Z 547.779,A -85,B 0,C 180,E1 -27094.434,E2 -27094.434} C_VEL
LIN {X 0,Y 91.2,Z 547.181,A -85,B 0,C 180,E1 -27098.865,E2 -27098.865} C_VEL
LIN {X 0,Y 93.062,Z 544.716,A -85,B 0,C 180,E1 -27107.581,E2 -27107.581} C_VEL
LIN {X 0,Y 95.703,Z 541.756,A -85,B 0,C 180,E1 -27113.821,E2 -27113.821} C_VEL
LIN {X 0,Y 99.434,Z 537.763,A -85,B 0,C 180,E1 -27119.652,E2 -27119.652} C_VEL
LIN {X 0,Y 104.112,Z 532.631,A -85,B 0,C 180,E1 -27125.013,E2 -27125.013} C_VEL
LIN {X 0,Y 107.933,Z 528.04,A -85,B 0,C 180,E1 -27128.705,E2 -27128.705} C_VEL
LIN {X 0,Y 112.384,Z 522.42,A -85,B 0,C 180,E1 -27132.24,E2 -27132.24} C_VEL
LIN {X 0,Y 114.404,Z 519.665,A -85,B 0,C 180,E1 -27133.716,E2 -27133.716} C_VEL
LIN {X 0,Y 116.366,Z 515.034,A -85,B 0,C 180,E1 -27136.446,E2 -27136.446} C_VEL
LIN {X 0,Y 118.502,Z 507.994,A -85,B 0,C 180,E1 -27140.441,E2 -27140.441} C_VEL
LIN {X 0,Y 119.978,Z 501.17,A -85,B 0,C 180,E1 -27144.14,E2 -27144.14} C_VEL
LIN {X 0,Y 120.354,Z 497.042,A -85,B 0,C 180,E1 -27146.493,E2 -27146.493} C_VEL
LIN {X 0,Y 119.904,Z 491.769,A -85,B 0,C 180,E1 -27150.118,E2 -27150.118} C_VEL
LIN {X 0,Y 119.08,Z 487.24,A -85,B 0,C 180,E1 -27153.725,E2 -27153.725} C_VEL
LIN {X 0,Y 118.078,Z 482.925,A -85,B 0,C 180,E1 -27157.609,E2 -27157.609} C_VEL
LIN {X 0,Y 117.267,Z 479.888,A -85,B 0,C 180,E1 -27160.752,E2 -27160.752} C_VEL
LIN {X 0,Y 116.081,Z 476.015,A -85,B 0,C 180,E1 -27165.983,E2 -27165.983} C_VEL
LIN {X 0,Y 115.361,Z 474.102,A -85,B 0,C 180,E1 -27169.467,E2 -27169.467} C_VEL
LIN {X 0,Y 114.512,Z 470.967,A -85,B 0,C 180,E1 -27179.998,E2 -27179.998} C_VEL
LIN {X 0,Y 114.95,Z 473.78,A -85,B 0,C 180,E1 -27190.567,E2 -27190.567} C_VEL
LIN {X 0,Y 115.652,Z 475.173,A -85,B 0,C 180,E1 -27194.066,E2 -27194.066} C_VEL
LIN {X 0,Y 116.947,Z 478.212,A -85,B 0,C 180,E1 -27199.299,E2 -27199.299} C_VEL
LIN {X 0,Y 118.674,Z 482.277,A -85,B 0,C 180,E1 -27204.489,E2 -27204.489} C_VEL
LIN {X 0,Y 119.949,Z 486.056,A -85,B 0,C 180,E1 -27208.496,E2 -27208.496} C_VEL
LIN {X 0,Y 121.637,Z 491.736,A -85,B 0,C 180,E1 -27213.539,E2 -27213.539} C_VEL
LIN {X 0,Y 122.731,Z 497.049,A -85,B 0,C 180,E1 -27217.723,E2 -27217.723} C_VEL
LIN {X 0,Y 123.502,Z 503.275,A -85,B 0,C 180,E1 -27222.29,E2 -27222.29} C_VEL
LIN {X 0,Y 123.649,Z 508.456,A -85,B 0,C 180,E1 -27225.925,E2 -27225.925} C_VEL
LIN {X 0,Y 123.528,Z 513.46,A -85,B 0,C 180,E1 -27229.467,E2 -27229.467} C_VEL
LIN {X 0,Y 123.276,Z 520.462,A -85,B 0,C 180,E1 -27235.038,E2 -27235.038} C_VEL
LIN {X 0,Y 122.76,Z 522.497,A -85,B 0,C 180,E1 -27236.645,E2 -27236.645} C_VEL
LIN {X 0,Y 120.45,Z 525.942,A -85,B 0,C 180,E1 -27239.178,E2 -27239.178} C_VEL
LIN {X 0,Y 118.467,Z 529.082,A -85,B 0,C 180,E1 -27241.866,E2 -27241.866} C_VEL
LIN {X 0,Y 118.471,Z 530.533,A -85,B 0,C 180,E1 -27243.638,E2 -27243.638} C_VEL
LIN {X 0,Y 121.974,Z 534.536,A -85,B 0,C 180,E1 -27249.776,E2 -27249.776} C_VEL
LIN {X 0,Y 125.322,Z 536.711,A -85,B 0,C 180,E1 -27253.717,E2 -27253.717} C_VEL
LIN {X 0,Y 129.534,Z 538.371,A -85,B 0,C 180,E1 -27257.575,E2 -27257.575} C_VEL
LIN {X 0,Y 139.63,Z 540.365,A -85,B 0,C 180,E1 -27264.223,E2 -27264.223} C_VEL
LIN {X 0,Y 147.658,Z 540.837,A -85,B 0,C 180,E1 -27268.185,E2 -27268.185} C_VEL
LIN {X 0,Y 151.924,Z 540.713,A -85,B 0,C 180,E1 -27270.001,E2 -27270.001} C_VEL
LIN {X 0,Y 145.567,Z 540.755,A -85,B 0,C 180,E1 -27272.768,E2 -27272.768} C_VEL
LIN {X 0,Y 139.623,Z 540.365,A -85,B 0,C 180,E1 -27275.778,E2 -27275.778} C_VEL
LIN {X 0,Y 129.381,Z 538.316,A -85,B 0,C 180,E1 -27282.55,E2 -27282.55} C_VEL
LIN {X 0,Y 124.807,Z 536.458,A -85,B 0,C 180,E1 -27286.814,E2 -27286.814} C_VEL
LIN {X 0,Y 120.98,Z 533.746,A -85,B 0,C 180,E1 -27291.652,E2 -27291.652} C_VEL
LIN {X 0,Y 117.686,Z 528.919,A -85,B 0,C 180,E1 -27298.539,E2 -27298.539} C_VEL
LIN {X 0,Y 116.532,Z 523.165,A -85,B 0,C 180,E1 -27304.956,E2 -27304.956} C_VEL
LIN {X 0,Y 116.965,Z 517.071,A -85,B 0,C 180,E1 -27310.417,E2 -27310.417} C_VEL
LIN {X 0,Y 117.438,Z 512.536,A -85,B 0,C 180,E1 -27314.102,E2 -27314.102} C_VEL
LIN {X 0,Y 117.582,Z 506.399,A -85,B 0,C 180,E1 -27318.895,E2 -27318.895} C_VEL
LIN {X 0,Y 117.037,Z 499.874,A -85,B 0,C 180,E1 -27324.165,E2 -27324.165} C_VEL
LIN {X 0,Y 116.006,Z 494.46,A -85,B 0,C 180,E1 -27329.006,E2 -27329.006} C_VEL
LIN {X 0,Y 115.214,Z 490.727,A -85,B 0,C 180,E1 -27332.777,E2 -27332.777} C_VEL
LIN {X 0,Y 113.735,Z 486.176,A -85,B 0,C 180,E1 -27338.24,E2 -27338.24} C_VEL
LIN {X 0,Y 112.575,Z 482.723,A -85,B 0,C 180,E1 -27343.686,E2 -27343.686} C_VEL
LIN {X 0,Y 111.615,Z 480.161,A -85,B 0,C 180,E1 -27349.113,E2 -27349.113} C_VEL
LIN {X 0,Y 111.416,Z 477.434,A -85,B 0,C 180,E1 -27360.002,E2 -27360.002} C_VEL
LIN {X 0,Y 112.027,Z 480.641,A -85,B 0,C 180,E1 -27370.85,E2 -27370.85} C_VEL
LIN {X 0,Y 112.892,Z 484.021,A -85,B 0,C 180,E1 -27376.271,E2 -27376.271} C_VEL
LIN {X 0,Y 113.276,Z 485.306,A -85,B 0,C 180,E1 -27378.074,E2 -27378.074} C_VEL
LIN {X 0,Y 113.941,Z 489.041,A -85,B 0,C 180,E1 -27382.299,E2 -27382.299} C_VEL
LIN {X 0,Y 114.833,Z 495.471,A -85,B 0,C 180,E1 -27388.109,E2 -27388.109} C_VEL
LIN {X 0,Y 114.983,Z 500.921,A -85,B 0,C 180,E1 -27392.269,E2 -27392.269} C_VEL
LIN {X 0,Y 114.181,Z 505.223,A -85,B 0,C 180,E1 -27394.914,E2 -27394.914} C_VEL
LIN {X 0,Y 112.246,Z 511.801,A -85,B 0,C 180,E1 -27398.767,E2 -27398.767} C_VEL
LIN {X 0,Y 109.828,Z 518.037,A -85,B 0,C 180,E1 -27402.617,E2 -27402.617} C_VEL
LIN {X 0,Y 108.286,Z 520.828,A -85,B 0,C 180,E1 -27404.444,E2 -27404.444} C_VEL
LIN {X 0,Y 103.144,Z 527.063,A -85,B 0,C 180,E1 -27408.271,E2 -27408.271} C_VEL
LIN {X 0,Y 98.353,Z 532.417,A -85,B 0,C 180,E1 -27412.599,E2 -27412.599} C_VEL
LIN {X 0,Y 93.29,Z 537.548,A -85,B 0,C 180,E1 -27418.173,E2 -27418.173} C_VEL
LIN {X 0,Y 89.219,Z 541.542,A -85,B 0,C 180,E1 -27424.325,E2 -27424.325} C_VEL
LIN {X 0,Y 86.293,Z 544.503,A -85,B 0,C 180,E1 -27430.987,E2 -27430.987} C_VEL
LIN {X 0,Y 84.177,Z 546.969,A -85,B 0,C 180,E1 -27440.387,E2 -27440.387} C_VEL
LIN {X 0,Y 83.801,Z 547.567,A -85,B 0,C 180,E1 -27445.188,E2 -27445.188} C_VEL
LIN {X 0,Y 83.883,Z 547.731,A -85,B 0,C 180,E1 -27449.999,E2 -27449.999} C_VEL
LIN {X 0,Y 83.801,Z 547.568,A -85,B 0,C 180,E1 -27454.81,E2 -27454.81} C_VEL
LIN {X 0,Y 84.176,Z 546.969,A -85,B 0,C 180,E1 -27459.611,E2 -27459.611} C_VEL
LIN {X 0,Y 86.292,Z 544.504,A -85,B 0,C 180,E1 -27469.011,E2 -27469.011} C_VEL
LIN {X 0,Y 89.217,Z 541.543,A -85,B 0,C 180,E1 -27475.673,E2 -27475.673} C_VEL
LIN {X 0,Y 93.286,Z 537.55,A -85,B 0,C 180,E1 -27481.826,E2 -27481.826} C_VEL
LIN {X 0,Y 98.347,Z 532.418,A -85,B 0,C 180,E1 -27487.402,E2 -27487.402} C_VEL
LIN {X 0,Y 104.069,Z 525.995,A -85,B 0,C 180,E1 -27492.477,E2 -27492.477} C_VEL
LIN {X 0,Y 108.282,Z 520.83,A -85,B 0,C 180,E1 -27495.555,E2 -27495.555} C_VEL
LIN {X 0,Y 109.861,Z 518.041,A -85,B 0,C 180,E1 -27497.362,E2 -27497.362} C_VEL
LIN {X 0,Y 112.658,Z 510.651,A -85,B 0,C 180,E1 -27501.95,E2 -27501.95} C_VEL
LIN {X 0,Y 114.773,Z 502.807,A -85,B 0,C 180,E1 -27506.555,E2 -27506.555} C_VEL
LIN {X 0,Y 114.98,Z 498.162,A -85,B 0,C 180,E1 -27509.715,E2 -27509.715} C_VEL
LIN {X 0,Y 114.694,Z 493.911,A -85,B 0,C 180,E1 -27513.227,E2 -27513.227} C_VEL
LIN {X 0,Y 113.85,Z 488.5,A -85,B 0,C 180,E1 -27518.259,E2 -27518.259} C_VEL
LIN {X 0,Y 113.277,Z 485.305,A -85,B 0,C 180,E1 -27521.926,E2 -27521.926} C_VEL
LIN {X 0,Y 112.297,Z 481.59,A -85,B 0,C 180,E1 -27527.345,E2 -27527.345} C_VEL
LIN {X 0,Y 112.026,Z 480.643,A -85,B 0,C 180,E1 -27529.15,E2 -27529.15} C_VEL
LIN {X 0,Y 111.418,Z 477.429,A -85,B 0,C 180,E1 -27539.998,E2 -27539.998} C_VEL
LIN {X 0,Y 111.613,Z 480.164,A -85,B 0,C 180,E1 -27550.887,E2 -27550.887} C_VEL
LIN {X 0,Y 112.213,Z 481.751,A -85,B 0,C 180,E1 -27554.506,E2 -27554.506} C_VEL
LIN {X 0,Y 113.311,Z 484.923,A -85,B 0,C 180,E1 -27559.944,E2 -27559.944} C_VEL
LIN {X 0,Y 114.703,Z 489.055,A -85,B 0,C 180,E1 -27565.396,E2 -27565.396} C_VEL
LIN {X 0,Y 115.593,Z 492.559,A -85,B 0,C 180,E1 -27569.102,E2 -27569.102} C_VEL
LIN {X 0,Y 116.715,Z 497.53,A -85,B 0,C 180,E1 -27573.845,E2 -27573.845} C_VEL
LIN {X 0,Y 117.402,Z 503.554,A -85,B 0,C 180,E1 -27578.905,E2 -27578.905} C_VEL
LIN {X 0,Y 117.581,Z 508.646,A -85,B 0,C 180,E1 -27582.933,E2 -27582.933} C_VEL
LIN {X 0,Y 117.229,Z 514.903,A -85,B 0,C 180,E1 -27587.832,E2 -27587.832} C_VEL
LIN {X 0,Y 116.614,Z 520.941,A -85,B 0,C 180,E1 -27592.94,E2 -27592.94} C_VEL
LIN {X 0,Y 116.824,Z 525.401,A -85,B 0,C 180,E1 -27597.372,E2 -27597.372} C_VEL
LIN {X 0,Y 118.471,Z 530.533,A -85,B 0,C 180,E1 -27603.638,E2 -27603.638} C_VEL
LIN {X 0,Y 119.093,Z 532.582,A -85,B 0,C 180,E1 -27606.326,E2 -27606.326} C_VEL
LIN {X 0,Y 119.239,Z 536.812,A -85,B 0,C 180,E1 -27612.692,E2 -27612.692} C_VEL
LIN {X 0,Y 120.574,Z 538.47,A -85,B 0,C 180,E1 -27616.289,E2 -27616.289} C_VEL
LIN {X 0,Y 122.064,Z 539.151,A -85,B 0,C 180,E1 -27617.961,E2 -27617.961} C_VEL
LIN {X 0,Y 130.172,Z 540.648,A -85,B 0,C 180,E1 -27623.802,E2 -27623.802} C_VEL
LIN {X 0,Y 140.567,Z 541.051,A -85,B 0,C 180,E1 -27629.262,E2 -27629.262} C_VEL
LIN {X 0,Y 142.248,Z 541.001,A -85,B 0,C 180,E1 -27630.001,E2 -27630.001} C_VEL
LIN {X 0,Y 133.865,Z 540.904,A -85,B 0,C 180,E1 -27634.068,E2 -27634.068} C_VEL
LIN {X 0,Y 124.939,Z 539.785,A -85,B 0,C 180,E1 -27639.716,E2 -27639.716} C_VEL
LIN {X 0,Y 120.446,Z 538.589,A -85,B 0,C 180,E1 -27643.498,E2 -27643.498} C_VEL
LIN {X 0,Y 115.083,Z 535.923,A -85,B 0,C 180,E1 -27649.626,E2 -27649.626} C_VEL
LIN {X 0,Y 112.57,Z 533.649,A -85,B 0,C 180,E1 -27653.94,E2 -27653.94} C_VEL
LIN {X 0,Y 110.353,Z 529.17,A -85,B 0,C 180,E1 -27660.631,E2 -27660.631} C_VEL
LIN {X 0,Y 109.901,Z 523.41,A -85,B 0,C 180,E1 -27667.41,E2 -27667.41} C_VEL
LIN {X 0,Y 110.844,Z 517.528,A -85,B 0,C 180,E1 -27672.968,E2 -27672.968} C_VEL
LIN {X 0,Y 111.486,Z 511.597,A -85,B 0,C 180,E1 -27678.171,E2 -27678.171} C_VEL
LIN {X 0,Y 111.568,Z 505.904,A -85,B 0,C 180,E1 -27683.247,E2 -27683.247} C_VEL
LIN {X 0,Y 111.162,Z 501.317,A -85,B 0,C 180,E1 -27687.545,E2 -27687.545} C_VEL
LIN {X 0,Y 110.378,Z 496.102,A -85,B 0,C 180,E1 -27693.051,E2 -27693.051} C_VEL
LIN {X 0,Y 109.673,Z 492.663,A -85,B 0,C 180,E1 -27697.39,E2 -27697.39} C_VEL
LIN {X 0,Y 108.68,Z 489.027,A -85,B 0,C 180,E1 -27703.084,E2 -27703.084} C_VEL
LIN {X 0,Y 107.934,Z 486.459,A -85,B 0,C 180,E1 -27708.737,E2 -27708.737} C_VEL
LIN {X 0,Y 107.602,Z 484.548,A -85,B 0,C 180,E1 -27716.257,E2 -27716.257} C_VEL
LIN {X 0,Y 108,Z 483.738,A -85,B 0,C 180,E1 -27720.002,E2 -27720.002} C_VEL
LIN {X 0,Y 107.953,Z 485.696,A -85,B 0,C 180,E1 -27727.484,E2 -27727.484} C_VEL
LIN {X 0,Y 108.378,Z 487.02,A -85,B 0,C 180,E1 -27731.22,E2 -27731.22} C_VEL
LIN {X 0,Y 108.95,Z 490.48,A -85,B 0,C 180,E1 -27736.877,E2 -27736.877} C_VEL
LIN {X 0,Y 109.356,Z 493.67,A -85,B 0,C 180,E1 -27740.702,E2 -27740.702} C_VEL
LIN {X 0,Y 109.713,Z 499.479,A -85,B 0,C 180,E1 -27746.644,E2 -27746.644} C_VEL
LIN {X 0,Y 109.682,Z 503.189,A -85,B 0,C 180,E1 -27749.777,E2 -27749.777} C_VEL
LIN {X 0,Y 109.074,Z 506.348,A -85,B 0,C 180,E1 -27752.105,E2 -27752.105} C_VEL
LIN {X 0,Y 107.621,Z 511.038,A -85,B 0,C 180,E1 -27755.079,E2 -27755.079} C_VEL
LIN {X 0,Y 104.768,Z 517.808,A -85,B 0,C 180,E1 -27759.517,E2 -27759.517} C_VEL
LIN {X 0,Y 103.258,Z 520.608,A -85,B 0,C 180,E1 -27761.523,E2 -27761.523} C_VEL
LIN {X 0,Y 98.928,Z 525.78,A -85,B 0,C 180,E1 -27764.731,E2 -27764.731} C_VEL
LIN {X 0,Y 94.731,Z 530.286,A -85,B 0,C 180,E1 -27768.11,E2 -27768.11} C_VEL
LIN {X 0,Y 89.009,Z 535.78,A -85,B 0,C 180,E1 -27773.687,E2 -27773.687} C_VEL
LIN {X 0,Y 84.232,Z 540.111,A -85,B 0,C 180,E1 -27779.959,E2 -27779.959} C_VEL
LIN {X 0,Y 81.591,Z 542.482,A -85,B 0,C 180,E1 -27784.488,E2 -27784.488} C_VEL
LIN {X 0,Y 79.593,Z 544.291,A -85,B 0,C 180,E1 -27789.316,E2 -27789.316} C_VEL
LIN {X 0,Y 77.183,Z 546.758,A -85,B 0,C 180,E1 -27799.506,E2 -27799.506} C_VEL
LIN {X 0,Y 76.739,Z 547.356,A -85,B 0,C 180,E1 -27804.744,E2 -27804.744} C_VEL
LIN {X 0,Y 76.782,Z 547.52,A -85,B 0,C 180,E1 -27809.999,E2 -27809.999} C_VEL
LIN {X 0,Y 76.739,Z 547.357,A -85,B 0,C 180,E1 -27815.253,E2 -27815.253} C_VEL
LIN {X 0,Y 77.183,Z 546.758,A -85,B 0,C 180,E1 -27820.492,E2 -27820.492} C_VEL
LIN {X 0,Y 79.592,Z 544.292,A -85,B 0,C 180,E1 -27830.682,E2 -27830.682} C_VEL
LIN {X 0,Y 82.849,Z 541.331,A -85,B 0,C 180,E1 -27837.809,E2 -27837.809} C_VEL
LIN {X 0,Y 87.295,Z 537.337,A -85,B 0,C 180,E1 -27844.301,E2 -27844.301} C_VEL
LIN {X 0,Y 92.772,Z 532.206,A -85,B 0,C 180,E1 -27850.083,E2 -27850.083} C_VEL
LIN {X 0,Y 97.74,Z 527.054,A -85,B 0,C 180,E1 -27854.367,E2 -27854.367} C_VEL
LIN {X 0,Y 102.258,Z 521.994,A -85,B 0,C 180,E1 -27857.63,E2 -27857.63} C_VEL
LIN {X 0,Y 103.279,Z 520.612,A -85,B 0,C 180,E1 -27858.462,E2 -27858.462} C_VEL
LIN {X 0,Y 105.469,Z 516.221,A -85,B 0,C 180,E1 -27861.531,E2 -27861.531} C_VEL
LIN {X 0,Y 108.194,Z 509.357,A -85,B 0,C 180,E1 -27866.003,E2 -27866.003} C_VEL
LIN {X 0,Y 109.477,Z 504.619,A -85,B 0,C 180,E1 -27869.096,E2 -27869.096} C_VEL
LIN {X 0,Y 109.749,Z 500.639,A -85,B 0,C 180,E1 -27872.335,E2 -27872.335} C_VEL
LIN {X 0,Y 109.463,Z 495.47,A -85,B 0,C 180,E1 -27877.34,E2 -27877.34} C_VEL
LIN {X 0,Y 109.391,Z 493.618,A -85,B 0,C 180,E1 -27879.305,E2 -27879.305} C_VEL
LIN {X 0,Y 108.947,Z 490.484,A -85,B 0,C 180,E1 -27883.123,E2 -27883.123} C_VEL
LIN {X 0,Y 108.376,Z 487.024,A -85,B 0,C 180,E1 -27888.78,E2 -27888.78} C_VEL
LIN {X 0,Y 107.956,Z 485.692,A -85,B 0,C 180,E1 -27892.517,E2 -27892.517} C_VEL
LIN {X 0,Y 108.002,Z 483.734,A -85,B 0,C 180,E1 -27899.998,E2 -27899.998} C_VEL
LIN {X 0,Y 107.925,Z 486.473,A -85,B 0,C 180,E1 -27911.264,E2 -27911.264} C_VEL
LIN {X 0,Y 108.668,Z 489.046,A -85,B 0,C 180,E1 -27916.918,E2 -27916.918} C_VEL
LIN {X 0,Y 109.697,Z 492.629,A -85,B 0,C 180,E1 -27922.605,E2 -27922.605} C_VEL
LIN {X 0,Y 110.393,Z 496.105,A -85,B 0,C 180,E1 -27926.968,E2 -27926.968} C_VEL
LIN {X 0,Y 111.248,Z 501.292,A -85,B 0,C 180,E1 -27932.506,E2 -27932.506} C_VEL
LIN {X 0,Y 111.636,Z 507.1,A -85,B 0,C 180,E1 -27937.862,E2 -27937.862} C_VEL
LIN {X 0,Y 111.416,Z 513.067,A -85,B 0,C 180,E1 -27943.058,E2 -27943.058} C_VEL
LIN {X 0,Y 110.615,Z 518.863,A -85,B 0,C 180,E1 -27948.159,E2 -27948.159} C_VEL
LIN {X 0,Y 109.925,Z 525.513,A -85,B 0,C 180,E1 -27954.873,E2 -27954.873} C_VEL
LIN {X 0,Y 110.716,Z 530.434,A -85,B 0,C 180,E1 -27961.132,E2 -27961.132} C_VEL
LIN {X 0,Y 112.543,Z 533.651,A -85,B 0,C 180,E1 -27966.055,E2 -27966.055} C_VEL
LIN {X 0,Y 117.395,Z 537.303,A -85,B 0,C 180,E1 -27973.3,E2 -27973.3} C_VEL
LIN {X 0,Y 122.064,Z 539.151,A -85,B 0,C 180,E1 -27977.961,E2 -27977.961} C_VEL
LIN {X 0,Y 123.392,Z 539.783,A -85,B 0,C 180,E1 -27979.698,E2 -27979.698} C_VEL
LIN {X 0,Y 125.522,Z 541.241,A -85,B 0,C 180,E1 -27985.8,E2 -27985.8} C_VEL
LIN {X 0,Y 127.44,Z 541.335,A -85,B 0,C 180,E1 -27987.375,E2 -27987.375} C_VEL
LIN {X 0,Y 132.592,Z 541.288,A -85,B 0,C 180,E1 -27990.001,E2 -27990.001} C_VEL
LIN {X 0,Y 126.421,Z 541.326,A -85,B 0,C 180,E1 -27993.187,E2 -27993.187} C_VEL
LIN {X 0,Y 120.362,Z 540.897,A -85,B 0,C 180,E1 -27996.973,E2 -27996.973} C_VEL
LIN {X 0,Y 111.652,Z 538.859,A -85,B 0,C 180,E1 -28004.584,E2 -28004.584} C_VEL
LIN {X 0,Y 108.198,Z 537.245,A -85,B 0,C 180,E1 -28008.952,E2 -28008.952} C_VEL
LIN {X 0,Y 104.756,Z 533.904,A -85,B 0,C 180,E1 -28015.855,E2 -28015.855} C_VEL
LIN {X 0,Y 103.192,Z 529.421,A -85,B 0,C 180,E1 -28023.015,E2 -28023.015} C_VEL
LIN {X 0,Y 103.547,Z 523.905,A -85,B 0,C 180,E1 -28029.861,E2 -28029.861} C_VEL
LIN {X 0,Y 104.66,Z 519.102,A -85,B 0,C 180,E1 -28034.837,E2 -28034.837} C_VEL
LIN {X 0,Y 105.572,Z 513.01,A -85,B 0,C 180,E1 -28040.776,E2 -28040.776} C_VEL
LIN {X 0,Y 105.735,Z 509.043,A -85,B 0,C 180,E1 -28044.675,E2 -28044.675} C_VEL
LIN {X 0,Y 105.755,Z 506.021,A -85,B 0,C 180,E1 -28047.886,E2 -28047.886} C_VEL
LIN {X 0,Y 105.348,Z 500.502,A -85,B 0,C 180,E1 -28054.304,E2 -28054.304} C_VEL
LIN {X 0,Y 104.63,Z 496.336,A -85,B 0,C 180,E1 -28060.378,E2 -28060.378} C_VEL
LIN {X 0,Y 104.251,Z 494.18,A -85,B 0,C 180,E1 -28064.358,E2 -28064.358} C_VEL
LIN {X 0,Y 103.973,Z 492.553,A -85,B 0,C 180,E1 -28068.302,E2 -28068.302} C_VEL
LIN {X 0,Y 103.7,Z 490.551,A -85,B 0,C 180,E1 -28076.116,E2 -28076.116} C_VEL
LIN {X 0,Y 104.106,Z 489.771,A -85,B 0,C 180,E1 -28080.002,E2 -28080.002} C_VEL
LIN {X 0,Y 104.04,Z 491.756,A -85,B 0,C 180,E1 -28087.767,E2 -28087.767} C_VEL
LIN {X 0,Y 104.369,Z 494.083,A -85,B 0,C 180,E1 -28093.08,E2 -28093.08} C_VEL
LIN {X 0,Y 104.489,Z 495.538,A -85,B 0,C 180,E1 -28095.609,E2 -28095.609} C_VEL
LIN {X 0,Y 104.567,Z 498.644,A -85,B 0,C 180,E1 -28099.789,E2 -28099.789} C_VEL
LIN {X 0,Y 104.54,Z 503.386,A -85,B 0,C 180,E1 -28105.01,E2 -28105.01} C_VEL
LIN {X 0,Y 104.146,Z 507.232,A -85,B 0,C 180,E1 -28108.685,E2 -28108.685} C_VEL
LIN {X 0,Y 102.981,Z 511.006,A -85,B 0,C 180,E1 -28111.457,E2 -28111.457} C_VEL
LIN {X 0,Y 99.956,Z 517.574,A -85,B 0,C 180,E1 -28116.042,E2 -28116.042} C_VEL
LIN {X 0,Y 97.521,Z 521.776,A -85,B 0,C 180,E1 -28119.22,E2 -28119.22} C_VEL
LIN {X 0,Y 90.185,Z 529.489,A -85,B 0,C 180,E1 -28124.539,E2 -28124.539} C_VEL
LIN {X 0,Y 83.38,Z 535.569,A -85,B 0,C 180,E1 -28130.789,E2 -28130.789} C_VEL
LIN {X 0,Y 78.139,Z 539.899,A -85,B 0,C 180,E1 -28137.339,E2 -28137.339} C_VEL
LIN {X 0,Y 75.214,Z 542.27,A -85,B 0,C 180,E1 -28142.147,E2 -28142.147} C_VEL
LIN {X 0,Y 72.96,Z 544.078,A -85,B 0,C 180,E1 -28147.336,E2 -28147.336} C_VEL
LIN {X 0,Y 70.194,Z 546.546,A -85,B 0,C 180,E1 -28158.448,E2 -28158.448} C_VEL
LIN {X 0,Y 69.655,Z 547.145,A -85,B 0,C 180,E1 -28164.208,E2 -28164.208} C_VEL
LIN {X 0,Y 69.703,Z 547.309,A -85,B 0,C 180,E1 -28169.999,E2 -28169.999} C_VEL
LIN {X 0,Y 69.655,Z 547.145,A -85,B 0,C 180,E1 -28175.79,E2 -28175.79} C_VEL
LIN {X 0,Y 70.193,Z 546.546,A -85,B 0,C 180,E1 -28181.55,E2 -28181.55} C_VEL
LIN {X 0,Y 72.959,Z 544.079,A -85,B 0,C 180,E1 -28192.661,E2 -28192.661} C_VEL
LIN {X 0,Y 76.618,Z 541.119,A -85,B 0,C 180,E1 -28200.296,E2 -28200.296} C_VEL
LIN {X 0,Y 81.494,Z 537.124,A -85,B 0,C 180,E1 -28207.132,E2 -28207.132} C_VEL
LIN {X 0,Y 87.427,Z 531.993,A -85,B 0,C 180,E1 -28213.099,E2 -28213.099} C_VEL
LIN {X 0,Y 92.767,Z 526.842,A -85,B 0,C 180,E1 -28217.454,E2 -28217.454} C_VEL
LIN {X 0,Y 97.52,Z 521.779,A -85,B 0,C 180,E1 -28220.778,E2 -28220.778} C_VEL
LIN {X 0,Y 100.497,Z 516.474,A -85,B 0,C 180,E1 -28224.737,E2 -28224.737} C_VEL
LIN {X 0,Y 103.664,Z 509.191,A -85,B 0,C 180,E1 -28229.832,E2 -28229.832} C_VEL
LIN {X 0,Y 104.37,Z 505.574,A -85,B 0,C 180,E1 -28232.796,E2 -28232.796} C_VEL
LIN {X 0,Y 104.609,Z 502.223,A -85,B 0,C 180,E1 -28236.225,E2 -28236.225} C_VEL
LIN {X 0,Y 104.607,Z 498.463,A -85,B 0,C 180,E1 -28240.369,E2 -28240.369} C_VEL
LIN {X 0,Y 104.487,Z 495.541,A -85,B 0,C 180,E1 -28244.39,E2 -28244.39} C_VEL
LIN {X 0,Y 104.328,Z 493.318,A -85,B 0,C 180,E1 -28248.338,E2 -28248.338} C_VEL
LIN {X 0,Y 104.026,Z 491.777,A -85,B 0,C 180,E1 -28252.232,E2 -28252.232} C_VEL
LIN {X 0,Y 104.118,Z 489.753,A -85,B 0,C 180,E1 -28259.998,E2 -28259.998} C_VEL
LIN {X 0,Y 103.7,Z 491.467,A -85,B 0,C 180,E1 -28267.866,E2 -28267.866} C_VEL
LIN {X 0,Y 103.959,Z 492.572,A -85,B 0,C 180,E1 -28271.699,E2 -28271.699} C_VEL
LIN {X 0,Y 104.399,Z 495.229,A -85,B 0,C 180,E1 -28277.632,E2 -28277.632} C_VEL
LIN {X 0,Y 105.16,Z 498.98,A -85,B 0,C 180,E1 -28283.638,E2 -28283.638} C_VEL
LIN {X 0,Y 105.443,Z 502.211,A -85,B 0,C 180,E1 -28287.809,E2 -28287.809} C_VEL
LIN {X 0,Y 105.792,Z 505.974,A -85,B 0,C 180,E1 -28292.101,E2 -28292.101} C_VEL
LIN {X 0,Y 105.706,Z 510.751,A -85,B 0,C 180,E1 -28297.079,E2 -28297.079} C_VEL
LIN {X 0,Y 105.219,Z 515.699,A -85,B 0,C 180,E1 -28301.905,E2 -28301.905} C_VEL
LIN {X 0,Y 104.363,Z 520.313,A -85,B 0,C 180,E1 -28306.352,E2 -28306.352} C_VEL
LIN {X 0,Y 103.316,Z 525.757,A -85,B 0,C 180,E1 -28312.252,E2 -28312.252} C_VEL
LIN {X 0,Y 103.501,Z 530.998,A -85,B 0,C 180,E1 -28319.388,E2 -28319.388} C_VEL
LIN {X 0,Y 105.62,Z 535.06,A -85,B 0,C 180,E1 -28326.47,E2 -28326.47} C_VEL
LIN {X 0,Y 109.973,Z 538.122,A -85,B 0,C 180,E1 -28333.448,E2 -28333.448} C_VEL
LIN {X 0,Y 115.909,Z 540.082,A -85,B 0,C 180,E1 -28339.601,E2 -28339.601} C_VEL
LIN {X 0,Y 120.807,Z 540.928,A -85,B 0,C 180,E1 -28343.319,E2 -28343.319} C_VEL
LIN {X 0,Y 127.44,Z 541.335,A -85,B 0,C 180,E1 -28347.375,E2 -28347.375} C_VEL
LIN {X 0,Y 127.948,Z 541.428,A -85,B 0,C 180,E1 -28348.17,E2 -28348.17} C_VEL
LIN {X 0,Y 127.273,Z 541.447,A -85,B 0,C 180,E1 -28349.265,E2 -28349.265} C_VEL
LIN {X 0,Y 125.001,Z 541.525,A -85,B 0,C 180,E1 -28350.671,E2 -28350.671} C_VEL
LIN {X 0,Y 115.201,Z 541.478,A -85,B 0,C 180,E1 -28354.654,E2 -28354.654} C_VEL
LIN {X 0,Y 114.169,Z 541.408,A -85,B 0,C 180,E1 -28355.295,E2 -28355.295} C_VEL
LIN {X 0,Y 106.838,Z 540.333,A -85,B 0,C 180,E1 -28361.382,E2 -28361.382} C_VEL
LIN {X 0,Y 102.545,Z 538.946,A -85,B 0,C 180,E1 -28366.371,E2 -28366.371} C_VEL
LIN {X 0,Y 98.943,Z 536.66,A -85,B 0,C 180,E1 -28372.577,E2 -28372.577} C_VEL
LIN {X 0,Y 96.615,Z 532.715,A -85,B 0,C 180,E1 -28380.611,E2 -28380.611} C_VEL
LIN {X 0,Y 96.476,Z 527.757,A -85,B 0,C 180,E1 -28388.374,E2 -28388.374} C_VEL
LIN {X 0,Y 98.194,Z 521.667,A -85,B 0,C 180,E1 -28395.703,E2 -28395.703} C_VEL
LIN {X 0,Y 99.326,Z 516.715,A -85,B 0,C 180,E1 -28401.108,E2 -28401.108} C_VEL
LIN {X 0,Y 99.922,Z 512.568,A -85,B 0,C 180,E1 -28405.762,E2 -28405.762} C_VEL
LIN {X 0,Y 100.083,Z 508.577,A -85,B 0,C 180,E1 -28410.56,E2 -28410.56} C_VEL
LIN {X 0,Y 100.077,Z 504.529,A -85,B 0,C 180,E1 -28415.914,E2 -28415.914} C_VEL
LIN {X 0,Y 99.82,Z 501.195,A -85,B 0,C 180,E1 -28421.531,E2 -28421.531} C_VEL
LIN {X 0,Y 99.519,Z 498.42,A -85,B 0,C 180,E1 -28427.771,E2 -28427.771} C_VEL
LIN {X 0,Y 99.365,Z 497.178,A -85,B 0,C 180,E1 -28431.974,E2 -28431.974} C_VEL
LIN {X 0,Y 99.938,Z 495.6,A -85,B 0,C 180,E1 -28440.002,E2 -28440.002} C_VEL
LIN {X 0,Y 99.71,Z 498.072,A -85,B 0,C 180,E1 -28449.326,E2 -28449.326} C_VEL
LIN {X 0,Y 99.845,Z 500.416,A -85,B 0,C 180,E1 -28454.265,E2 -28454.265} C_VEL
LIN {X 0,Y 99.566,Z 504.034,A -85,B 0,C 180,E1 -28459.519,E2 -28459.519} C_VEL
LIN {X 0,Y 99.09,Z 508.846,A -85,B 0,C 180,E1 -28465.188,E2 -28465.188} C_VEL
LIN {X 0,Y 98.526,Z 511.042,A -85,B 0,C 180,E1 -28467.323,E2 -28467.323} C_VEL
LIN {X 0,Y 96.614,Z 515.205,A -85,B 0,C 180,E1 -28470.613,E2 -28470.613} C_VEL
LIN {X 0,Y 92.853,Z 521.547,A -85,B 0,C 180,E1 -28475.544,E2 -28475.544} C_VEL
LIN {X 0,Y 91.926,Z 522.942,A -85,B 0,C 180,E1 -28476.606,E2 -28476.606} C_VEL
LIN {X 0,Y 84.644,Z 529.861,A -85,B 0,C 180,E1 -28481.645,E2 -28481.645} C_VEL
LIN {X 0,Y 77.997,Z 535.357,A -85,B 0,C 180,E1 -28487.483,E2 -28487.483} C_VEL
LIN {X 0,Y 72.242,Z 539.687,A -85,B 0,C 180,E1 -28494.288,E2 -28494.288} C_VEL
LIN {X 0,Y 68.991,Z 542.058,A -85,B 0,C 180,E1 -28499.379,E2 -28499.379} C_VEL
LIN {X 0,Y 66.439,Z 543.866,A -85,B 0,C 180,E1 -28504.967,E2 -28504.967} C_VEL
LIN {X 0,Y 63.222,Z 546.334,A -85,B 0,C 180,E1 -28517.153,E2 -28517.153} C_VEL
LIN {X 0,Y 62.585,Z 546.933,A -85,B 0,C 180,E1 -28523.551,E2 -28523.551} C_VEL
LIN {X 0,Y 62.613,Z 547.098,A -85,B 0,C 180,E1 -28529.999,E2 -28529.999} C_VEL
LIN {X 0,Y 62.585,Z 546.933,A -85,B 0,C 180,E1 -28536.446,E2 -28536.446} C_VEL
LIN {X 0,Y 63.221,Z 546.334,A -85,B 0,C 180,E1 -28542.844,E2 -28542.844} C_VEL
LIN {X 0,Y 66.438,Z 543.867,A -85,B 0,C 180,E1 -28555.031,E2 -28555.031} C_VEL
LIN {X 0,Y 70.56,Z 540.907,A -85,B 0,C 180,E1 -28563.215,E2 -28563.215} C_VEL
LIN {X 0,Y 75.927,Z 536.912,A -85,B 0,C 180,E1 -28570.384,E2 -28570.384} C_VEL
LIN {X 0,Y 81.728,Z 532.326,A -85,B 0,C 180,E1 -28575.946,E2 -28575.946} C_VEL
LIN {X 0,Y 88.224,Z 526.514,A -85,B 0,C 180,E1 -28580.956,E2 -28580.956} C_VEL
LIN {X 0,Y 91.928,Z 522.945,A -85,B 0,C 180,E1 -28583.39,E2 -28583.39} C_VEL
LIN {X 0,Y 95.928,Z 516.526,A -85,B 0,C 180,E1 -28588.447,E2 -28588.447} C_VEL
LIN {X 0,Y 97.802,Z 512.738,A -85,B 0,C 180,E1 -28591.259,E2 -28591.259} C_VEL
LIN {X 0,Y 98.893,Z 509.879,A -85,B 0,C 180,E1 -28593.785,E2 -28593.785} C_VEL
LIN {X 0,Y 99.305,Z 506.906,A -85,B 0,C 180,E1 -28596.927,E2 -28596.927} C_VEL
LIN {X 0,Y 99.717,Z 502.853,A -85,B 0,C 180,E1 -28602.044,E2 -28602.044} C_VEL
LIN {X 0,Y 99.842,Z 500.42,A -85,B 0,C 180,E1 -28605.735,E2 -28605.735} C_VEL
LIN {X 0,Y 99.824,Z 499.275,A -85,B 0,C 180,E1 -28607.804,E2 -28607.804} C_VEL
LIN {X 0,Y 99.691,Z 497.62,A -85,B 0,C 180,E1 -28611.892,E2 -28611.892} C_VEL
LIN {X 0,Y 99.955,Z 495.577,A -85,B 0,C 180,E1 -28619.998,E2 -28619.998} C_VEL
LIN {X 0,Y 99.368,Z 497.201,A -85,B 0,C 180,E1 -28628.13,E2 -28628.13} C_VEL
LIN {X 0,Y 99.517,Z 498.423,A -85,B 0,C 180,E1 -28632.229,E2 -28632.229} C_VEL
LIN {X 0,Y 99.808,Z 501.208,A -85,B 0,C 180,E1 -28638.471,E2 -28638.471} C_VEL
LIN {X 0,Y 100.031,Z 503.618,A -85,B 0,C 180,E1 -28642.732,E2 -28642.732} C_VEL
LIN {X 0,Y 100.144,Z 506.817,A -85,B 0,C 180,E1 -28647.137,E2 -28647.137} C_VEL
LIN {X 0,Y 100.041,Z 511.046,A -85,B 0,C 180,E1 -28652.543,E2 -28652.543} C_VEL
LIN {X 0,Y 99.54,Z 515.561,A -85,B 0,C 180,E1 -28657.613,E2 -28657.613} C_VEL
LIN {X 0,Y 98.753,Z 519.531,A -85,B 0,C 180,E1 -28661.851,E2 -28661.851} C_VEL
LIN {X 0,Y 96.943,Z 526.002,A -85,B 0,C 180,E1 -28669.274,E2 -28669.274} C_VEL
LIN {X 0,Y 96.407,Z 531.245,A -85,B 0,C 180,E1 -28676.858,E2 -28676.858} C_VEL
LIN {X 0,Y 97.826,Z 535.315,A -85,B 0,C 180,E1 -28684.467,E2 -28684.467} C_VEL
LIN {X 0,Y 99.929,Z 537.507,A -85,B 0,C 180,E1 -28689.413,E2 -28689.413} C_VEL
LIN {X 0,Y 102.954,Z 539.128,A -85,B 0,C 180,E1 -28694.155,E2 -28694.155} C_VEL
LIN {X 0,Y 111.516,Z 541.207,A -85,B 0,C 180,E1 -28702.76,E2 -28702.76} C_VEL
LIN {X 0,Y 122.021,Z 541.603,A -85,B 0,C 180,E1 -28709.471,E2 -28709.471} C_VEL
LIN {X 0,Y 123.018,Z 541.573,A -85,B 0,C 180,E1 -28710.001,E2 -28710.001} C_VEL
LIN {X 0,Y 114.169,Z 541.408,A -85,B 0,C 180,E1 -28715.295,E2 -28715.295} C_VEL
LIN {X 0,Y 110.303,Z 541.204,A -85,B 0,C 180,E1 -28717.58,E2 -28717.58} C_VEL
LIN {X 0,Y 97.595,Z 540.125,A -85,B 0,C 180,E1 -28724.462,E2 -28724.462} C_VEL
LIN {X 0,Y 94.5,Z 539.358,A -85,B 0,C 180,E1 -28727.402,E2 -28727.402} C_VEL
LIN {X 0,Y 93.781,Z 539.014,A -85,B 0,C 180,E1 -28728.491,E2 -28728.491} C_VEL
LIN {X 0,Y 90.911,Z 536.696,A -85,B 0,C 180,E1 -28735.172,E2 -28735.172} C_VEL
LIN {X 0,Y 89.741,Z 534.449,A -85,B 0,C 180,E1 -28740.525,E2 -28740.525} C_VEL
LIN {X 0,Y 89.739,Z 529.914,A -85,B 0,C 180,E1 -28748.795,E2 -28748.795} C_VEL
LIN {X 0,Y 91.605,Z 524.453,A -85,B 0,C 180,E1 -28756.335,E2 -28756.335} C_VEL
LIN {X 0,Y 93.295,Z 519.124,A -85,B 0,C 180,E1 -28762.943,E2 -28762.943} C_VEL
LIN {X 0,Y 94.22,Z 514.729,A -85,B 0,C 180,E1 -28768.527,E2 -28768.527} C_VEL
LIN {X 0,Y 94.516,Z 511.155,A -85,B 0,C 180,E1 -28773.506,E2 -28773.506} C_VEL
LIN {X 0,Y 94.804,Z 508.17,A -85,B 0,C 180,E1 -28778.246,E2 -28778.246} C_VEL
LIN {X 0,Y 94.783,Z 505.828,A -85,B 0,C 180,E1 -28782.749,E2 -28782.749} C_VEL
LIN {X 0,Y 94.726,Z 504.044,A -85,B 0,C 180,E1 -28787.142,E2 -28787.142} C_VEL
LIN {X 0,Y 94.74,Z 502.792,A -85,B 0,C 180,E1 -28791.47,E2 -28791.47} C_VEL
LIN {X 0,Y 95.495,Z 501.24,A -85,B 0,C 180,E1 -28800.002,E2 -28800.002} C_VEL
LIN {X 0,Y 95.077,Z 503.259,A -85,B 0,C 180,E1 -28808.504,E2 -28808.504} C_VEL
LIN {X 0,Y 94.948,Z 505.052,A -85,B 0,C 180,E1 -28812.832,E2 -28812.832} C_VEL
LIN {X 0,Y 94.542,Z 507.778,A -85,B 0,C 180,E1 -28817.301,E2 -28817.301} C_VEL
LIN {X 0,Y 93.702,Z 511.929,A -85,B 0,C 180,E1 -28822.943,E2 -28822.943} C_VEL
LIN {X 0,Y 93.132,Z 513.821,A -85,B 0,C 180,E1 -28825.102,E2 -28825.102} C_VEL
LIN {X 0,Y 91.093,Z 517.6,A -85,B 0,C 180,E1 -28828.304,E2 -28828.304} C_VEL
LIN {X 0,Y 87.574,Z 522.714,A -85,B 0,C 180,E1 -28832.578,E2 -28832.578} C_VEL
LIN {X 0,Y 86.538,Z 523.986,A -85,B 0,C 180,E1 -28833.65,E2 -28833.65} C_VEL
LIN {X 0,Y 79.649,Z 529.985,A -85,B 0,C 180,E1 -28838.149,E2 -28838.149} C_VEL
LIN {X 0,Y 72.913,Z 535.145,A -85,B 0,C 180,E1 -28843.704,E2 -28843.704} C_VEL
LIN {X 0,Y 66.589,Z 539.475,A -85,B 0,C 180,E1 -28850.708,E2 -28850.708} C_VEL
LIN {X 0,Y 62.966,Z 541.846,A -85,B 0,C 180,E1 -28856.076,E2 -28856.076} C_VEL
LIN {X 0,Y 60.039,Z 543.654,A -85,B 0,C 180,E1 -28862.079,E2 -28862.079} C_VEL
LIN {X 0,Y 56.304,Z 546.122,A -85,B 0,C 180,E1 -28875.542,E2 -28875.542} C_VEL
LIN {X 0,Y 55.539,Z 546.722,A -85,B 0,C 180,E1 -28882.729,E2 -28882.729} C_VEL
LIN {X 0,Y 55.512,Z 546.887,A -85,B 0,C 180,E1 -28889.998,E2 -28889.998} C_VEL
LIN {X 0,Y 55.539,Z 546.722,A -85,B 0,C 180,E1 -28897.268,E2 -28897.268} C_VEL
LIN {X 0,Y 56.303,Z 546.122,A -85,B 0,C 180,E1 -28904.455,E2 -28904.455} C_VEL
LIN {X 0,Y 60.037,Z 543.654,A -85,B 0,C 180,E1 -28917.918,E2 -28917.918} C_VEL
LIN {X 0,Y 64.723,Z 540.695,A -85,B 0,C 180,E1 -28926.669,E2 -28926.669} C_VEL
LIN {X 0,Y 70.649,Z 536.7,A -85,B 0,C 180,E1 -28934.131,E2 -28934.131} C_VEL
LIN {X 0,Y 76.607,Z 532.376,A -85,B 0,C 180,E1 -28939.504,E2 -28939.504} C_VEL
LIN {X 0,Y 82.614,Z 527.458,A -85,B 0,C 180,E1 -28943.915,E2 -28943.915} C_VEL
LIN {X 0,Y 86.539,Z 523.988,A -85,B 0,C 180,E1 -28946.345,E2 -28946.345} C_VEL
LIN {X 0,Y 90.274,Z 518.78,A -85,B 0,C 180,E1 -28950.701,E2 -28950.701} C_VEL
LIN {X 0,Y 92.156,Z 515.818,A -85,B 0,C 180,E1 -28953.174,E2 -28953.174} C_VEL
LIN {X 0,Y 93.136,Z 513.824,A -85,B 0,C 180,E1 -28954.889,E2 -28954.889} C_VEL
LIN {X 0,Y 93.9,Z 511.164,A -85,B 0,C 180,E1 -28958.021,E2 -28958.021} C_VEL
LIN {X 0,Y 94.57,Z 507.746,A -85,B 0,C 180,E1 -28962.704,E2 -28962.704} C_VEL
LIN {X 0,Y 94.948,Z 505.052,A -85,B 0,C 180,E1 -28967.168,E2 -28967.168} C_VEL
LIN {X 0,Y 95.083,Z 503.252,A -85,B 0,C 180,E1 -28971.497,E2 -28971.497} C_VEL
LIN {X 0,Y 95.523,Z 501.208,A -85,B 0,C 180,E1 -28979.998,E2 -28979.998} C_VEL
LIN {X 0,Y 94.738,Z 502.794,A -85,B 0,C 180,E1 -28988.53,E2 -28988.53} C_VEL
LIN {X 0,Y 94.748,Z 505.001,A -85,B 0,C 180,E1 -28995.365,E2 -28995.365} C_VEL
LIN {X 0,Y 94.847,Z 506.919,A -85,B 0,C 180,E1 -28999.475,E2 -28999.475} C_VEL
LIN {X 0,Y 94.718,Z 509.523,A -85,B 0,C 180,E1 -29004.082,E2 -29004.082} C_VEL
LIN {X 0,Y 94.457,Z 512.813,A -85,B 0,C 180,E1 -29008.917,E2 -29008.917} C_VEL
LIN {X 0,Y 94.035,Z 515.763,A -85,B 0,C 180,E1 -29012.892,E2 -29012.892} C_VEL
LIN {X 0,Y 93.084,Z 520.143,A -85,B 0,C 180,E1 -29018.29,E2 -29018.29} C_VEL
LIN {X 0,Y 91.584,Z 524.472,A -85,B 0,C 180,E1 -29023.678,E2 -29023.678} C_VEL
LIN {X 0,Y 89.8,Z 530.076,A -85,B 0,C 180,E1 -29031.497,E2 -29031.497} C_VEL
LIN {X 0,Y 89.747,Z 534.445,A -85,B 0,C 180,E1 -29039.469,E2 -29039.469} C_VEL
LIN {X 0,Y 91.791,Z 537.768,A -85,B 0,C 180,E1 -29047.493,E2 -29047.493} C_VEL
LIN {X 0,Y 95.155,Z 539.737,A -85,B 0,C 180,E1 -29053.763,E2 -29053.763} C_VEL
LIN {X 0,Y 102.389,Z 541.481,A -85,B 0,C 180,E1 -29062.11,E2 -29062.11} C_VEL
LIN {X 0,Y 107.575,Z 541.888,A -85,B 0,C 180,E1 -29066.255,E2 -29066.255} C_VEL
LIN {X 0,Y 113.523,Z 541.856,A -85,B 0,C 180,E1 -29070.001,E2 -29070.001} C_VEL
LIN {X 0,Y 105.825,Z 541.756,A -85,B 0,C 180,E1 -29075.042,E2 -29075.042} C_VEL
LIN {X 0,Y 97.971,Z 540.602,A -85,B 0,C 180,E1 -29082.428,E2 -29082.428} C_VEL
LIN {X 0,Y 93.781,Z 539.014,A -85,B 0,C 180,E1 -29088.491,E2 -29088.491} C_VEL
LIN {X 0,Y 91.482,Z 538.072,A -85,B 0,C 180,E1 -29091.809,E2 -29091.809} C_VEL
LIN {X 0,Y 83.78,Z 535.002,A -85,B 0,C 180,E1 -29102.147,E2 -29102.147} C_VEL
LIN {X 0,Y 82.71,Z 533.471,A -85,B 0,C 180,E1 -29105.977,E2 -29105.977} C_VEL
LIN {X 0,Y 82.706,Z 532.843,A -85,B 0,C 180,E1 -29107.264,E2 -29107.264} C_VEL
LIN {X 0,Y 84.303,Z 528.321,A -85,B 0,C 180,E1 -29115.122,E2 -29115.122} C_VEL
LIN {X 0,Y 85.595,Z 525.776,A -85,B 0,C 180,E1 -29118.942,E2 -29118.942} C_VEL
LIN {X 0,Y 87.015,Z 522.181,A -85,B 0,C 180,E1 -29123.87,E2 -29123.87} C_VEL
LIN {X 0,Y 88.112,Z 518.739,A -85,B 0,C 180,E1 -29128.777,E2 -29128.777} C_VEL
LIN {X 0,Y 88.939,Z 514.907,A -85,B 0,C 180,E1 -29134.942,E2 -29134.942} C_VEL
LIN {X 0,Y 89.414,Z 511.761,A -85,B 0,C 180,E1 -29140.598,E2 -29140.598} C_VEL
LIN {X 0,Y 89.666,Z 509.419,A -85,B 0,C 180,E1 -29146.403,E2 -29146.403} C_VEL
LIN {X 0,Y 89.822,Z 508.166,A -85,B 0,C 180,E1 -29151,E2 -29151} C_VEL
LIN {X 0,Y 90.639,Z 506.535,A -85,B 0,C 180,E1 -29160.002,E2 -29160.002} C_VEL
LIN {X 0,Y 90.242,Z 507.474,A -85,B 0,C 180,E1 -29164.469,E2 -29164.469} C_VEL
LIN {X 0,Y 90.084,Z 508.738,A -85,B 0,C 180,E1 -29168.979,E2 -29168.979} C_VEL
LIN {X 0,Y 89.642,Z 510.698,A -85,B 0,C 180,E1 -29173.606,E2 -29173.606} C_VEL
LIN {X 0,Y 88.767,Z 513.611,A -85,B 0,C 180,E1 -29178.466,E2 -29178.466} C_VEL
LIN {X 0,Y 87.89,Z 516.416,A -85,B 0,C 180,E1 -29182.326,E2 -29182.326} C_VEL
LIN {X 0,Y 87.189,Z 517.68,A -85,B 0,C 180,E1 -29183.771,E2 -29183.771} C_VEL
LIN {X 0,Y 83.621,Z 522.481,A -85,B 0,C 180,E1 -29188.056,E2 -29188.056} C_VEL
LIN {X 0,Y 81.39,Z 524.93,A -85,B 0,C 180,E1 -29190.288,E2 -29190.288} C_VEL
LIN {X 0,Y 74.836,Z 530.218,A -85,B 0,C 180,E1 -29194.3,E2 -29194.3} C_VEL
LIN {X 0,Y 68.192,Z 534.933,A -85,B 0,C 180,E1 -29199.378,E2 -29199.378} C_VEL
LIN {X 0,Y 61.246,Z 539.263,A -85,B 0,C 180,E1 -29206.487,E2 -29206.487} C_VEL
LIN {X 0,Y 57.2,Z 541.634,A -85,B 0,C 180,E1 -29212.095,E2 -29212.095} C_VEL
LIN {X 0,Y 51.216,Z 544.839,A -85,B 0,C 180,E1 -29225.689,E2 -29225.689} C_VEL
LIN {X 0,Y 49.453,Z 545.91,A -85,B 0,C 180,E1 -29233.486,E2 -29233.486} C_VEL
LIN {X 0,Y 48.497,Z 546.51,A -85,B 0,C 180,E1 -29241.666,E2 -29241.666} C_VEL
LIN {X 0,Y 48.43,Z 546.676,A -85,B 0,C 180,E1 -29249.998,E2 -29249.998} C_VEL
LIN {X 0,Y 48.496,Z 546.511,A -85,B 0,C 180,E1 -29258.331,E2 -29258.331} C_VEL
LIN {X 0,Y 49.453,Z 545.91,A -85,B 0,C 180,E1 -29266.511,E2 -29266.511} C_VEL
LIN {X 0,Y 53.828,Z 543.442,A -85,B 0,C 180,E1 -29281.481,E2 -29281.481} C_VEL
LIN {X 0,Y 59.17,Z 540.484,A -85,B 0,C 180,E1 -29290.786,E2 -29290.786} C_VEL
LIN {X 0,Y 65.726,Z 536.488,A -85,B 0,C 180,E1 -29298.458,E2 -29298.458} C_VEL
LIN {X 0,Y 72.929,Z 531.573,A -85,B 0,C 180,E1 -29304.446,E2 -29304.446} C_VEL
LIN {X 0,Y 79.995,Z 526.089,A -85,B 0,C 180,E1 -29308.932,E2 -29308.932} C_VEL
LIN {X 0,Y 81.387,Z 524.932,A -85,B 0,C 180,E1 -29309.712,E2 -29309.712} C_VEL
LIN {X 0,Y 83.607,Z 522.483,A -85,B 0,C 180,E1 -29311.957,E2 -29311.957} C_VEL
LIN {X 0,Y 87.111,Z 517.747,A -85,B 0,C 180,E1 -29316.207,E2 -29316.207} C_VEL
LIN {X 0,Y 88.294,Z 515.341,A -85,B 0,C 180,E1 -29319.008,E2 -29319.008} C_VEL
LIN {X 0,Y 89.232,Z 512.179,A -85,B 0,C 180,E1 -29323.708,E2 -29323.708} C_VEL
LIN {X 0,Y 89.643,Z 510.698,A -85,B 0,C 180,E1 -29326.394,E2 -29326.394} C_VEL
LIN {X 0,Y 90.085,Z 508.737,A -85,B 0,C 180,E1 -29331.021,E2 -29331.021} C_VEL
LIN {X 0,Y 90.257,Z 507.458,A -85,B 0,C 180,E1 -29335.532,E2 -29335.532} C_VEL
LIN {X 0,Y 90.669,Z 506.502,A -85,B 0,C 180,E1 -29339.998,E2 -29339.998} C_VEL
LIN {X 0,Y 89.82,Z 508.168,A -85,B 0,C 180,E1 -29349.001,E2 -29349.001} C_VEL
LIN {X 0,Y 89.645,Z 509.439,A -85,B 0,C 180,E1 -29353.601,E2 -29353.601} C_VEL
LIN {X 0,Y 89.425,Z 511.762,A -85,B 0,C 180,E1 -29359.427,E2 -29359.427} C_VEL
LIN {X 0,Y 88.967,Z 514.897,A -85,B 0,C 180,E1 -29365.08,E2 -29365.08} C_VEL
LIN {X 0,Y 88.127,Z 518.725,A -85,B 0,C 180,E1 -29371.217,E2 -29371.217} C_VEL
LIN {X 0,Y 87.045,Z 522.182,A -85,B 0,C 180,E1 -29376.16,E2 -29376.16} C_VEL
LIN {X 0,Y 85.239,Z 526.488,A -85,B 0,C 180,E1 -29382.096,E2 -29382.096} C_VEL
LIN {X 0,Y 83.246,Z 531.142,A -85,B 0,C 180,E1 -29389.444,E2 -29389.444} C_VEL
LIN {X 0,Y 82.712,Z 535.351,A -85,B 0,C 180,E1 -29398.173,E2 -29398.173} C_VEL
LIN {X 0,Y 84.322,Z 538.363,A -85,B 0,C 180,E1 -29406.459,E2 -29406.459} C_VEL
LIN {X 0,Y 87.74,Z 540.417,A -85,B 0,C 180,E1 -29413.977,E2 -29413.977} C_VEL
LIN {X 0,Y 93.382,Z 541.752,A -85,B 0,C 180,E1 -29421.344,E2 -29421.344} C_VEL
LIN {X 0,Y 98.615,Z 542.182,A -85,B 0,C 180,E1 -29426.108,E2 -29426.108} C_VEL
LIN {X 0,Y 104.081,Z 542.137,A -85,B 0,C 180,E1 -29430.001,E2 -29430.001} C_VEL
LIN {X 0,Y 98.359,Z 542.162,A -85,B 0,C 180,E1 -29434.098,E2 -29434.098} C_VEL
LIN {X 0,Y 92.623,Z 541.67,A -85,B 0,C 180,E1 -29439.474,E2 -29439.474} C_VEL
LIN {X 0,Y 86.11,Z 539.652,A -85,B 0,C 180,E1 -29449.055,E2 -29449.055} C_VEL
LIN {X 0,Y 83.264,Z 536.954,A -85,B 0,C 180,E1 -29457.662,E2 -29457.662} C_VEL
LIN {X 0,Y 82.655,Z 533.213,A -85,B 0,C 180,E1 -29466.527,E2 -29466.527} C_VEL
LIN {X 0,Y 82.706,Z 532.843,A -85,B 0,C 180,E1 -29467.264,E2 -29467.264} C_VEL
LIN {X 0,Y 82.626,Z 531.058,A -85,B 0,C 180,E1 -29471.165,E2 -29471.165} C_VEL
LIN {X 0,Y 81.616,Z 528.132,A -85,B 0,C 180,E1 -29477.757,E2 -29477.757} C_VEL
LIN {X 0,Y 81.132,Z 524.447,A -85,B 0,C 180,E1 -29485.81,E2 -29485.81} C_VEL
LIN {X 0,Y 81.619,Z 522.932,A -85,B 0,C 180,E1 -29488.407,E2 -29488.407} C_VEL
LIN {X 0,Y 82.666,Z 520.342,A -85,B 0,C 180,E1 -29492.91,E2 -29492.91} C_VEL
LIN {X 0,Y 83.442,Z 517.637,A -85,B 0,C 180,E1 -29497.894,E2 -29497.894} C_VEL
LIN {X 0,Y 83.791,Z 516.466,A -85,B 0,C 180,E1 -29500.4,E2 -29500.4} C_VEL
LIN {X 0,Y 84.205,Z 514.602,A -85,B 0,C 180,E1 -29505.502,E2 -29505.502} C_VEL
LIN {X 0,Y 84.478,Z 513.181,A -85,B 0,C 180,E1 -29510.425,E2 -29510.425} C_VEL
LIN {X 0,Y 84.867,Z 512.215,A -85,B 0,C 180,E1 -29515.252,E2 -29515.252} C_VEL
LIN {X 0,Y 85.516,Z 511.556,A -85,B 0,C 180,E1 -29520.003,E2 -29520.003} C_VEL
LIN {X 0,Y 84.878,Z 512.93,A -85,B 0,C 180,E1 -29526.477,E2 -29526.477} C_VEL
LIN {X 0,Y 84.339,Z 514.873,A -85,B 0,C 180,E1 -29532.027,E2 -29532.027} C_VEL
LIN {X 0,Y 83.863,Z 516.164,A -85,B 0,C 180,E1 -29534.564,E2 -29534.564} C_VEL
LIN {X 0,Y 82.329,Z 519.414,A -85,B 0,C 180,E1 -29540.114,E2 -29540.114} C_VEL
LIN {X 0,Y 81.579,Z 520.496,A -85,B 0,C 180,E1 -29541.363,E2 -29541.363} C_VEL
LIN {X 0,Y 77.833,Z 524.704,A -85,B 0,C 180,E1 -29545.449,E2 -29545.449} C_VEL
LIN {X 0,Y 76.552,Z 525.874,A -85,B 0,C 180,E1 -29546.476,E2 -29546.476} C_VEL
LIN {X 0,Y 68.451,Z 531.761,A -85,B 0,C 180,E1 -29551.12,E2 -29551.12} C_VEL
LIN {X 0,Y 61.244,Z 536.275,A -85,B 0,C 180,E1 -29556.554,E2 -29556.554} C_VEL
LIN {X 0,Y 53.968,Z 540.27,A -85,B 0,C 180,E1 -29564.254,E2 -29564.254} C_VEL
LIN {X 0,Y 47.884,Z 543.228,A -85,B 0,C 180,E1 -29574.048,E2 -29574.048} C_VEL
LIN {X 0,Y 42.662,Z 545.698,A -85,B 0,C 180,E1 -29590.762,E2 -29590.762} C_VEL
LIN {X 0,Y 41.47,Z 546.299,A -85,B 0,C 180,E1 -29600.241,E2 -29600.241} C_VEL
LIN {X 0,Y 41.33,Z 546.465,A -85,B 0,C 180,E1 -29609.998,E2 -29609.998} C_VEL
LIN {X 0,Y 41.47,Z 546.299,A -85,B 0,C 180,E1 -29619.755,E2 -29619.755} C_VEL
LIN {X 0,Y 42.661,Z 545.698,A -85,B 0,C 180,E1 -29629.235,E2 -29629.235} C_VEL
LIN {X 0,Y 47.883,Z 543.229,A -85,B 0,C 180,E1 -29645.949,E2 -29645.949} C_VEL
LIN {X 0,Y 53.965,Z 540.271,A -85,B 0,C 180,E1 -29655.745,E2 -29655.745} C_VEL
LIN {X 0,Y 61.239,Z 536.276,A -85,B 0,C 180,E1 -29663.447,E2 -29663.447} C_VEL
LIN {X 0,Y 68.262,Z 531.881,A -85,B 0,C 180,E1 -29668.784,E2 -29668.784} C_VEL
LIN {X 0,Y 75.097,Z 527.033,A -85,B 0,C 180,E1 -29672.752,E2 -29672.752} C_VEL
LIN {X 0,Y 76.552,Z 525.876,A -85,B 0,C 180,E1 -29673.519,E2 -29673.519} C_VEL
LIN {X 0,Y 78.988,Z 523.525,A -85,B 0,C 180,E1 -29675.779,E2 -29675.779} C_VEL
LIN {X 0,Y 81.567,Z 520.485,A -85,B 0,C 180,E1 -29678.682,E2 -29678.682} C_VEL
LIN {X 0,Y 82.396,Z 519.297,A -85,B 0,C 180,E1 -29680.048,E2 -29680.048} C_VEL
LIN {X 0,Y 83.914,Z 516.119,A -85,B 0,C 180,E1 -29685.445,E2 -29685.445} C_VEL
LIN {X 0,Y 84.337,Z 514.875,A -85,B 0,C 180,E1 -29687.973,E2 -29687.973} C_VEL
LIN {X 0,Y 84.884,Z 512.935,A -85,B 0,C 180,E1 -29693.469,E2 -29693.469} C_VEL
LIN {X 0,Y 85.548,Z 511.527,A -85,B 0,C 180,E1 -29699.997,E2 -29699.997} C_VEL
LIN {X 0,Y 84.471,Z 513.188,A -85,B 0,C 180,E1 -29709.576,E2 -29709.576} C_VEL
LIN {X 0,Y 84.196,Z 514.61,A -85,B 0,C 180,E1 -29714.499,E2 -29714.499} C_VEL
LIN {X 0,Y 83.82,Z 516.442,A -85,B 0,C 180,E1 -29719.593,E2 -29719.593} C_VEL
LIN {X 0,Y 82.997,Z 519.174,A -85,B 0,C 180,E1 -29725.046,E2 -29725.046} C_VEL
LIN {X 0,Y 81.837,Z 522.462,A -85,B 0,C 180,E1 -29730.823,E2 -29730.823} C_VEL
LIN {X 0,Y 80.4,Z 525.75,A -85,B 0,C 180,E1 -29736.047,E2 -29736.047} C_VEL
LIN {X 0,Y 77.748,Z 530.399,A -85,B 0,C 180,E1 -29743.687,E2 -29743.687} C_VEL
LIN {X 0,Y 75.886,Z 534.908,A -85,B 0,C 180,E1 -29752.99,E2 -29752.99} C_VEL
LIN {X 0,Y 76.274,Z 538.277,A -85,B 0,C 180,E1 -29762.569,E2 -29762.569} C_VEL
LIN {X 0,Y 80.337,Z 541.019,A -85,B 0,C 180,E1 -29774.206,E2 -29774.206} C_VEL
LIN {X 0,Y 85.294,Z 542.096,A -85,B 0,C 180,E1 -29781.387,E2 -29781.387} C_VEL
LIN {X 0,Y 91.451,Z 542.515,A -85,B 0,C 180,E1 -29787.446,E2 -29787.446} C_VEL
LIN {X 0,Y 94.783,Z 542.414,A -85,B 0,C 180,E1 -29790.001,E2 -29790.001} C_VEL
LIN {X 0,Y 89.227,Z 542.435,A -85,B 0,C 180,E1 -29794.519,E2 -29794.519} C_VEL
LIN {X 0,Y 84.481,Z 542.02,A -85,B 0,C 180,E1 -29799.578,E2 -29799.578} C_VEL
LIN {X 0,Y 77.963,Z 539.91,A -85,B 0,C 180,E1 -29811.137,E2 -29811.137} C_VEL
LIN {X 0,Y 75.861,Z 537.3,A -85,B 0,C 180,E1 -29820.383,E2 -29820.383} C_VEL
LIN {X 0,Y 75.898,Z 534.467,A -85,B 0,C 180,E1 -29828.026,E2 -29828.026} C_VEL
LIN {X 0,Y 77.724,Z 530.399,A -85,B 0,C 180,E1 -29836.335,E2 -29836.335} C_VEL
LIN {X 0,Y 80.384,Z 525.749,A -85,B 0,C 180,E1 -29843.973,E2 -29843.973} C_VEL
LIN {X 0,Y 81.619,Z 522.932,A -85,B 0,C 180,E1 -29848.407,E2 -29848.407} C_VEL
LIN {X 0,Y 81.987,Z 521.602,A -85,B 0,C 180,E1 -29850.975,E2 -29850.975} C_VEL
LIN {X 0,Y 81.628,Z 520.18,A -85,B 0,C 180,E1 -29854.997,E2 -29854.997} C_VEL
LIN {X 0,Y 80.687,Z 519.304,A -85,B 0,C 180,E1 -29859.125,E2 -29859.125} C_VEL
LIN {X 0,Y 78.912,Z 517.717,A -85,B 0,C 180,E1 -29870.953,E2 -29870.953} C_VEL
LIN {X 0,Y 79.399,Z 516.975,A -85,B 0,C 180,E1 -29874.925,E2 -29874.925} C_VEL
LIN {X 0,Y 80.144,Z 516.36,A -85,B 0,C 180,E1 -29880.003,E2 -29880.003} C_VEL
LIN {X 0,Y 79.553,Z 517.273,A -85,B 0,C 180,E1 -29885.071,E2 -29885.071} C_VEL
LIN {X 0,Y 78.743,Z 519.016,A -85,B 0,C 180,E1 -29890.955,E2 -29890.955} C_VEL
LIN {X 0,Y 77.445,Z 521.374,A -85,B 0,C 180,E1 -29895.801,E2 -29895.801} C_VEL
LIN {X 0,Y 76.857,Z 522.42,A -85,B 0,C 180,E1 -29897.64,E2 -29897.64} C_VEL
LIN {X 0,Y 73.487,Z 525.648,A -85,B 0,C 180,E1 -29901.179,E2 -29901.179} C_VEL
LIN {X 0,Y 72.111,Z 526.818,A -85,B 0,C 180,E1 -29902.197,E2 -29902.197} C_VEL
LIN {X 0,Y 63.061,Z 532.846,A -85,B 0,C 180,E1 -29906.927,E2 -29906.927} C_VEL
LIN {X 0,Y 54.502,Z 537.595,A -85,B 0,C 180,E1 -29913.051,E2 -29913.051} C_VEL
LIN {X 0,Y 46.8,Z 541.211,A -85,B 0,C 180,E1 -29921.334,E2 -29921.334} C_VEL
LIN {X 0,Y 42.314,Z 543.016,A -85,B 0,C 180,E1 -29928.364,E2 -29928.364} C_VEL
LIN {X 0,Y 36.014,Z 545.486,A -85,B 0,C 180,E1 -29947.025,E2 -29947.025} C_VEL
LIN {X 0,Y 34.492,Z 546.087,A -85,B 0,C 180,E1 -29958.241,E2 -29958.241} C_VEL
LIN {X 0,Y 34.245,Z 546.254,A -85,B 0,C 180,E1 -29969.997,E2 -29969.997} C_VEL
LIN {X 0,Y 34.491,Z 546.087,A -85,B 0,C 180,E1 -29981.754,E2 -29981.754} C_VEL
LIN {X 0,Y 36.013,Z 545.486,A -85,B 0,C 180,E1 -29992.97,E2 -29992.97} C_VEL
LIN {X 0,Y 42.312,Z 543.017,A -85,B 0,C 180,E1 -30011.633,E2 -30011.633} C_VEL
LIN {X 0,Y 49.255,Z 540.059,A -85,B 0,C 180,E1 -30021.696,E2 -30021.696} C_VEL
LIN {X 0,Y 57.289,Z 536.065,A -85,B 0,C 180,E1 -30029.17,E2 -30029.17} C_VEL
LIN {X 0,Y 65.969,Z 530.962,A -85,B 0,C 180,E1 -30034.773,E2 -30034.773} C_VEL
LIN {X 0,Y 72.107,Z 526.82,A -85,B 0,C 180,E1 -30037.804,E2 -30037.804} C_VEL
LIN {X 0,Y 74.752,Z 524.468,A -85,B 0,C 180,E1 -30040.075,E2 -30040.075} C_VEL
LIN {X 0,Y 76.868,Z 522.409,A -85,B 0,C 180,E1 -30042.37,E2 -30042.37} C_VEL
LIN {X 0,Y 78.326,Z 519.857,A -85,B 0,C 180,E1 -30047.037,E2 -30047.037} C_VEL
LIN {X 0,Y 78.851,Z 518.772,A -85,B 0,C 180,E1 -30049.729,E2 -30049.729} C_VEL
LIN {X 0,Y 79.553,Z 517.273,A -85,B 0,C 180,E1 -30054.929,E2 -30054.929} C_VEL
LIN {X 0,Y 80.174,Z 516.337,A -85,B 0,C 180,E1 -30059.997,E2 -30059.997} C_VEL
LIN {X 0,Y 79.069,Z 517.409,A -85,B 0,C 180,E1 -30067.406,E2 -30067.406} C_VEL
LIN {X 0,Y 78.747,Z 518.127,A -85,B 0,C 180,E1 -30070.981,E2 -30070.981} C_VEL
LIN {X 0,Y 78.097,Z 520.323,A -85,B 0,C 180,E1 -30078.356,E2 -30078.356} C_VEL
LIN {X 0,Y 76.981,Z 522.775,A -85,B 0,C 180,E1 -30084.088,E2 -30084.088} C_VEL
LIN {X 0,Y 75.583,Z 525.662,A -85,B 0,C 180,E1 -30089.803,E2 -30089.803} C_VEL
LIN {X 0,Y 73.907,Z 528.315,A -85,B 0,C 180,E1 -30094.785,E2 -30094.785} C_VEL
LIN {X 0,Y 71.242,Z 532.121,A -85,B 0,C 180,E1 -30101.989,E2 -30101.989} C_VEL
LIN {X 0,Y 68.985,Z 536.317,A -85,B 0,C 180,E1 -30112.321,E2 -30112.321} C_VEL
LIN {X 0,Y 68.891,Z 538.528,A -85,B 0,C 180,E1 -30119.333,E2 -30119.333} C_VEL
LIN {X 0,Y 69.965,Z 540.169,A -85,B 0,C 180,E1 -30126.311,E2 -30126.311} C_VEL
LIN {X 0,Y 75.747,Z 542.284,A -85,B 0,C 180,E1 -30139.307,E2 -30139.307} C_VEL
LIN {X 0,Y 84.345,Z 542.725,A -85,B 0,C 180,E1 -30149,E2 -30149} C_VEL
LIN {X 0,Y 85.533,Z 542.689,A -85,B 0,C 180,E1 -30150.001,E2 -30150.001} C_VEL
LIN {X 0,Y 77.982,Z 542.513,A -85,B 0,C 180,E1 -30157.562,E2 -30157.562} C_VEL
LIN {X 0,Y 72.305,Z 541.391,A -85,B 0,C 180,E1 -30166.955,E2 -30166.955} C_VEL
LIN {X 0,Y 69.718,Z 539.883,A -85,B 0,C 180,E1 -30174.88,E2 -30174.88} C_VEL
LIN {X 0,Y 68.779,Z 537.144,A -85,B 0,C 180,E1 -30185.175,E2 -30185.175} C_VEL
LIN {X 0,Y 70.167,Z 533.7,A -85,B 0,C 180,E1 -30194.518,E2 -30194.518} C_VEL
LIN {X 0,Y 73.094,Z 529.488,A -85,B 0,C 180,E1 -30203.085,E2 -30203.085} C_VEL
LIN {X 0,Y 74.803,Z 526.998,A -85,B 0,C 180,E1 -30207.735,E2 -30207.735} C_VEL
LIN {X 0,Y 76.18,Z 524.421,A -85,B 0,C 180,E1 -30212.534,E2 -30212.534} C_VEL
LIN {X 0,Y 77.561,Z 521.557,A -85,B 0,C 180,E1 -30218.752,E2 -30218.752} C_VEL
LIN {X 0,Y 78.071,Z 520.344,A -85,B 0,C 180,E1 -30221.638,E2 -30221.638} C_VEL
LIN {X 0,Y 78.839,Z 517.943,A -85,B 0,C 180,E1 -30229.733,E2 -30229.733} C_VEL
LIN {X 0,Y 78.912,Z 517.717,A -85,B 0,C 180,E1 -30230.953,E2 -30230.953} C_VEL
LIN {X 0,Y 78.641,Z 517.654,A -85,B 0,C 180,E1 -30233.787,E2 -30233.787} C_VEL
LIN {X 0,Y 77.703,Z 518.277,A -85,B 0,C 180,E1 -30236.575,E2 -30236.575} C_VEL
LIN {X 0,Y 73.535,Z 522.043,A -85,B 0,C 180,E1 -30246.154,E2 -30246.154} C_VEL
LIN {X 0,Y 72.577,Z 523.523,A -85,B 0,C 180,E1 -30251.17,E2 -30251.17} C_VEL
LIN {X 0,Y 71.542,Z 524.839,A -85,B 0,C 180,E1 -30254.217,E2 -30254.217} C_VEL
LIN {X 0,Y 69.586,Z 526.591,A -85,B 0,C 180,E1 -30256.366,E2 -30256.366} C_VEL
LIN {X 0,Y 68.119,Z 527.762,A -85,B 0,C 180,E1 -30257.379,E2 -30257.379} C_VEL
LIN {X 0,Y 57.066,Z 534.297,A -85,B 0,C 180,E1 -30262.53,E2 -30262.53} C_VEL
LIN {X 0,Y 48.037,Z 538.626,A -85,B 0,C 180,E1 -30268.617,E2 -30268.617} C_VEL
LIN {X 0,Y 42.425,Z 540.998,A -85,B 0,C 180,E1 -30274.074,E2 -30274.074} C_VEL
LIN {X 0,Y 37.283,Z 542.803,A -85,B 0,C 180,E1 -30281.058,E2 -30281.058} C_VEL
LIN {X 0,Y 29.597,Z 545.274,A -85,B 0,C 180,E1 -30301.643,E2 -30301.643} C_VEL
LIN {X 0,Y 27.56,Z 545.875,A -85,B 0,C 180,E1 -30315.223,E2 -30315.223} C_VEL
LIN {X 0,Y 27.132,Z 546.042,A -85,B 0,C 180,E1 -30329.997,E2 -30329.997} C_VEL
LIN {X 0,Y 27.56,Z 545.876,A -85,B 0,C 180,E1 -30344.771,E2 -30344.771} C_VEL
